PROGRAM P2_06_Device_Ctrl
VAR
	fbMixer_Motor					:FB_MotorFreqCtrl;
	fbMixerMotor_Speed				:FB_AnalogOutput_v01;
	fbSieve_Motor					:FB_MotorFreqCtrl;
	fbSieveMotor_Speed				:FB_AnalogOutput_v01;
	fbChopper_Motor					:FB_MotorCoilsCtrl;
	fbPump_Motor					:FB_CoilCtrl;
	
	fbSP_Temperature_PID			:FB_PID;
	
	fbSP_Mixer_Motor				:FB_MotorFreqCtrl;
	fbSP_MixerMotor_Speed			:FB_AnalogOutput_v01;
	fbSP_Pressure					:FB_AnalogOutput_v02;
	
	fbOutlet_Valve					:FB_ValveCtrl52;
	fbLid_Valve						:FB_ValveCtrl52;
	fbSieveSeal_Valve				:FB_ValveCtrl52;
	fbPurge_Valve					:FB_ValveCtrl52;
	fbTool_Valve					:FB_ValveCtrl52;
	
	fbCleaningAir_Valve				:FB_ValveCtrl32;
	fbPurifiedWater_Valve			:FB_ValveCtrl32;
	fbWarmWater_Valve				:FB_ValveCtrl32;
	fbColdWater_Valve				:FB_ValveCtrl32;
	fbMixerWIP_Valve				:FB_ValveCtrl32;
	fbChopperWIP_Valve				:FB_ValveCtrl32;
	fbSPWIP_Valve					:FB_ValveCtrl32;
	fbSPWIPDrain_Valve				:FB_ValveCtrl32;
	fbMainDrain_Valve				:FB_ValveCtrl32;
	
	fbAspiration_Valve				:FB_ValveCtrl32;
	fbVacuum_Valve					:FB_ValveCtrl32;
	fbFilterClean_Valve				:FB_ValveCtrl32;
	fbAirSeal_Valve					:FB_ValveCtrl32;
	fbMixerAir_Valve				:FB_ValveCtrl32;
	fbChopperAir_Valve				:FB_ValveCtrl32;
	
	
	
	

END_VAR

VAR PERSISTENT
	stMixer_Motor_Int				:ST_Interface_MotorCtrl;
	stSieve_Motor_Int				:ST_Interface_MotorCtrl;
	stChopper_Motor_Int				:ST_Interface_MotorCoilsCtrl;
	stPump_Motor_Int				:ST_Interface_CoilCtrl;
	
	stSP_Mixer_Motor_Int			:ST_Interface_MotorCtrl;
	stSP_Temperature_Int			:ST_Interface_PidCtrl;
	
	stOutlet_Valve_Int				:ST_Interface_ValveCtrl;
	stLid_Valve_Int					:ST_Interface_ValveCtrl;
	stSeal_Valve_Int				:ST_Interface_ValveCtrl;
	stPurge_Valve_Int				:ST_Interface_ValveCtrl;
	stTool_Valve_Int				:ST_Interface_ValveCtrl;
	
	stCleaningAir_Valve_INT			:ST_Interface_ValveCtrl;
	stPurifiedWater_Valve_INT		:ST_Interface_ValveCtrl;
	stWarmWater_Valve_Int			:ST_Interface_ValveCtrl;
	stColdWater_Valve_Int			:ST_Interface_ValveCtrl;
	stMixerWIP_Valve_Int			:ST_Interface_ValveCtrl;
	stChopperWIP_Valve_Int			:ST_Interface_ValveCtrl;
	stSPWIP_Valve_Int				:ST_Interface_ValveCtrl;
	stSPWIPDrain_Valve_Int			:ST_Interface_ValveCtrl;
	stMainDrain_Valve_Int			:ST_Interface_ValveCtrl;
	
	stAspiration_Valve_Int			:ST_Interface_ValveCtrl;
	stVacuum_Valve_Int				:ST_Interface_ValveCtrl;
	stFilterClean_Valve_Int			:ST_Interface_ValveCtrl;
	stAirSeal_Valve_Int				:ST_Interface_ValveCtrl;
	stMixerAir_Valve_Int			:ST_Interface_ValveCtrl;
	stChopperAir_Valve_Int			:ST_Interface_ValveCtrl;
END_VAR
VAR // added by the converter: edge detectors and wires of the graphical bodies
    _w1, _w2, _w3, _w4, _w5, _w6, _w7, _w8, _w9, _w10 : BOOL;
    _rt1, _rt2 : R_TRIG;
END_VAR

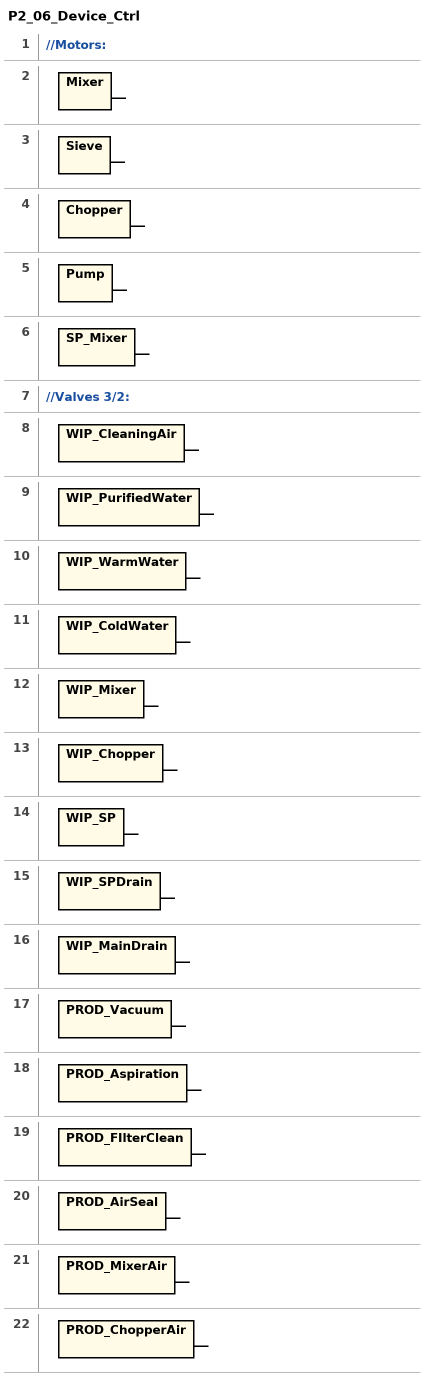
// NETWORK 1
// label: //Motors

// NETWORK 2
Mixer();

// NETWORK 3
Sieve();

// NETWORK 4
Chopper();

// NETWORK 5
Pump();

// NETWORK 6
SP_Mixer();

// NETWORK 7
// label: //Valves 3/2

// NETWORK 8
WIP_CleaningAir();

// NETWORK 9
WIP_PurifiedWater();

// NETWORK 10
WIP_WarmWater();

// NETWORK 11
WIP_ColdWater();

// NETWORK 12
WIP_Mixer();

// NETWORK 13
WIP_Chopper();

// NETWORK 14
WIP_SP();

// NETWORK 15
WIP_SPDrain();

// NETWORK 16
WIP_MainDrain();

// NETWORK 17
PROD_Vacuum();

// NETWORK 18
PROD_Aspiration();

// NETWORK 19
PROD_FIlterClean();

// NETWORK 20
PROD_AirSeal();

// NETWORK 21
PROD_MixerAir();

// NETWORK 22
PROD_ChopperAir();

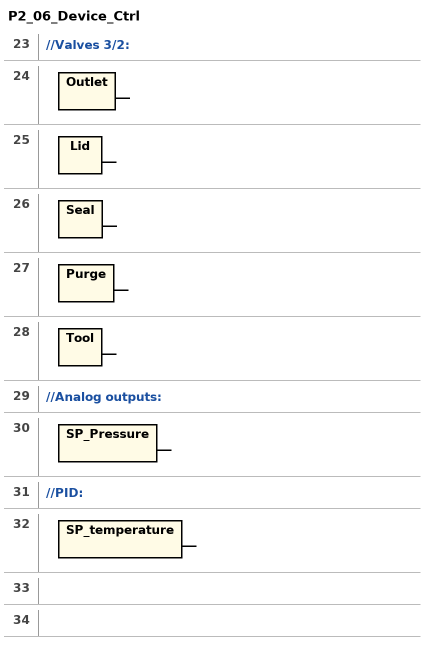
// NETWORK 23
// label: //Valves 3/2

// NETWORK 24
Outlet();

// NETWORK 25
Lid();

// NETWORK 26
Seal();

// NETWORK 27
Purge();

// NETWORK 28
Tool();

// NETWORK 29
// label: //Analog outputs

// NETWORK 30
SP_Pressure();

// NETWORK 31
// label: //PID

// NETWORK 32
SP_temperature();

// NETWORK 33

// NETWORK 34

ACTION Chopper:
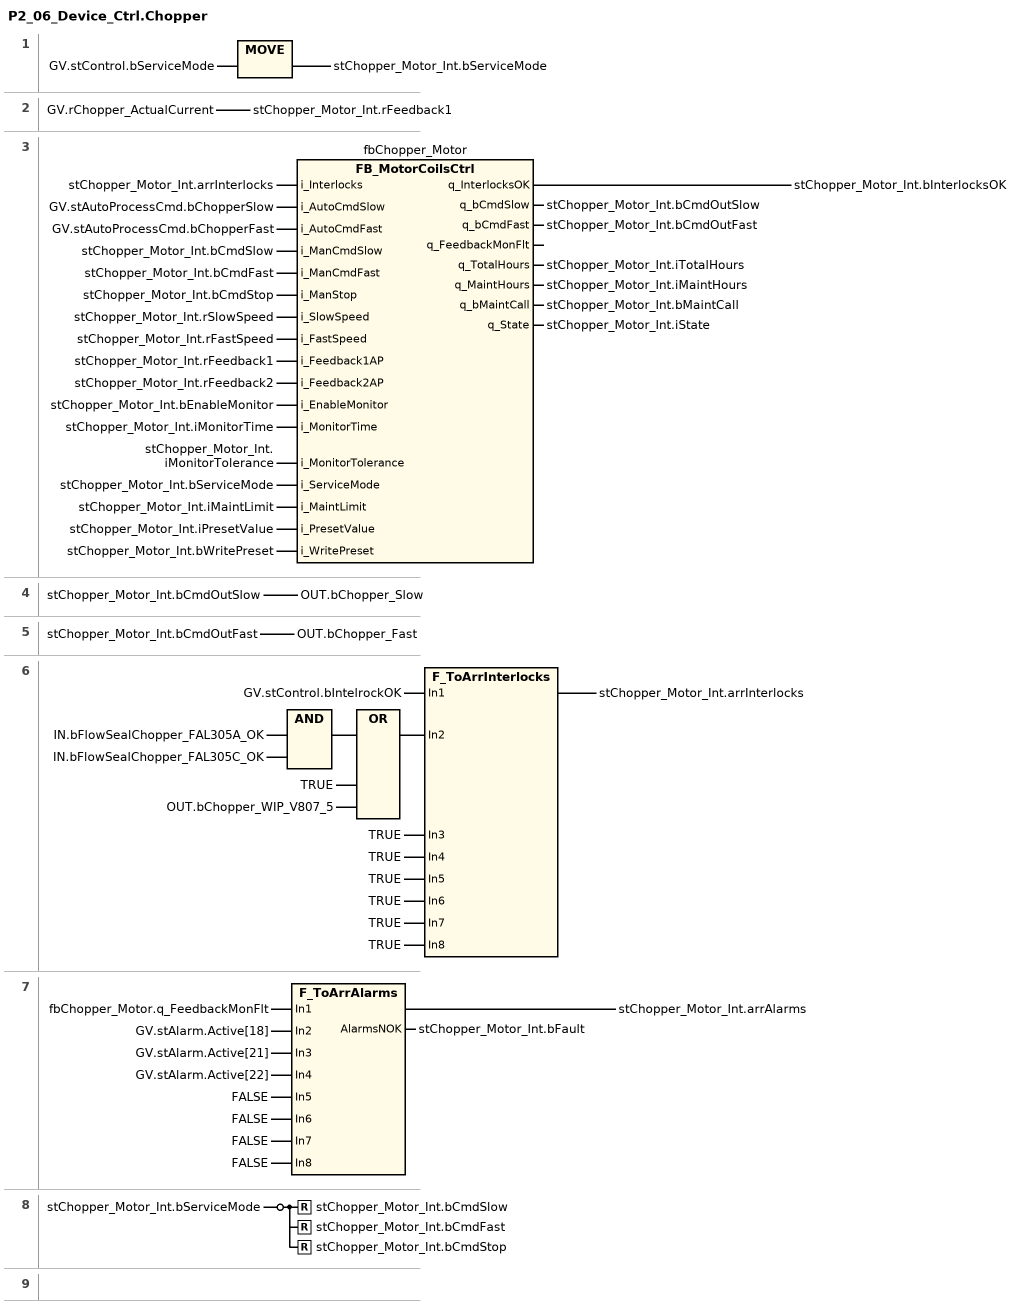
// NETWORK 1
stChopper_Motor_Int.bServiceMode := GV.stControl.bServiceMode;

// NETWORK 2
stChopper_Motor_Int.rFeedback1 := GV.rChopper_ActualCurrent;

// NETWORK 3
fbChopper_Motor(
    i_Interlocks := stChopper_Motor_Int.arrInterlocks,
    i_AutoCmdSlow := GV.stAutoProcessCmd.bChopperSlow,
    i_AutoCmdFast := GV.stAutoProcessCmd.bChopperFast,
    i_ManCmdSlow := stChopper_Motor_Int.bCmdSlow,
    i_ManCmdFast := stChopper_Motor_Int.bCmdFast,
    i_ManStop := stChopper_Motor_Int.bCmdStop,
    i_SlowSpeed := stChopper_Motor_Int.rSlowSpeed,
    i_FastSpeed := stChopper_Motor_Int.rFastSpeed,
    i_Feedback1AP := stChopper_Motor_Int.rFeedback1,
    i_Feedback2AP := stChopper_Motor_Int.rFeedback2,
    i_EnableMonitor := stChopper_Motor_Int.bEnableMonitor,
    i_MonitorTime := stChopper_Motor_Int.iMonitorTime,
    i_MonitorTolerance := stChopper_Motor_Int.iMonitorTolerance,
    i_ServiceMode := stChopper_Motor_Int.bServiceMode,
    i_MaintLimit := stChopper_Motor_Int.iMaintLimit,
    i_PresetValue := stChopper_Motor_Int.iPresetValue,
    i_WritePreset := stChopper_Motor_Int.bWritePreset,
    q_bCmdSlow => stChopper_Motor_Int.bCmdOutSlow,
    q_bCmdFast => stChopper_Motor_Int.bCmdOutFast,
    q_TotalHours => stChopper_Motor_Int.iTotalHours,
    q_MaintHours => stChopper_Motor_Int.iMaintHours,
    q_bMaintCall => stChopper_Motor_Int.bMaintCall,
    q_State => stChopper_Motor_Int.iState); // FB_MotorCoilsCtrl
stChopper_Motor_Int.bInterlocksOK := fbChopper_Motor.q_InterlocksOK;

// NETWORK 4
OUT.bChopper_Slow := stChopper_Motor_Int.bCmdOutSlow;

// NETWORK 5
OUT.bChopper_Fast := stChopper_Motor_Int.bCmdOutFast;

// NETWORK 6
stChopper_Motor_Int.arrInterlocks := F_ToArrInterlocks(In1 := GV.stControl.bIntelrockOK, In2 := IN.bFlowSealChopper_FAL305A_OK AND IN.bFlowSealChopper_FAL305C_OK OR TRUE OR OUT.bChopper_WIP_V807_5, In3 := TRUE, In4 := TRUE, In5 := TRUE, In6 := TRUE, In7 := TRUE, In8 := TRUE);

// NETWORK 7
stChopper_Motor_Int.arrAlarms := F_ToArrAlarms(In1 := fbChopper_Motor.q_FeedbackMonFlt, In2 := GV.stAlarm.Active[18], In3 := GV.stAlarm.Active[21], In4 := GV.stAlarm.Active[22], In5 := FALSE, In6 := FALSE, In7 := FALSE, In8 := FALSE, AlarmsNOK => stChopper_Motor_Int.bFault);

// NETWORK 8
_w1 := NOT stChopper_Motor_Int.bServiceMode;
stChopper_Motor_Int.bCmdSlow R= _w1;
stChopper_Motor_Int.bCmdFast R= _w1;
stChopper_Motor_Int.bCmdStop R= _w1;

// NETWORK 9
END_ACTION

ACTION Lid:
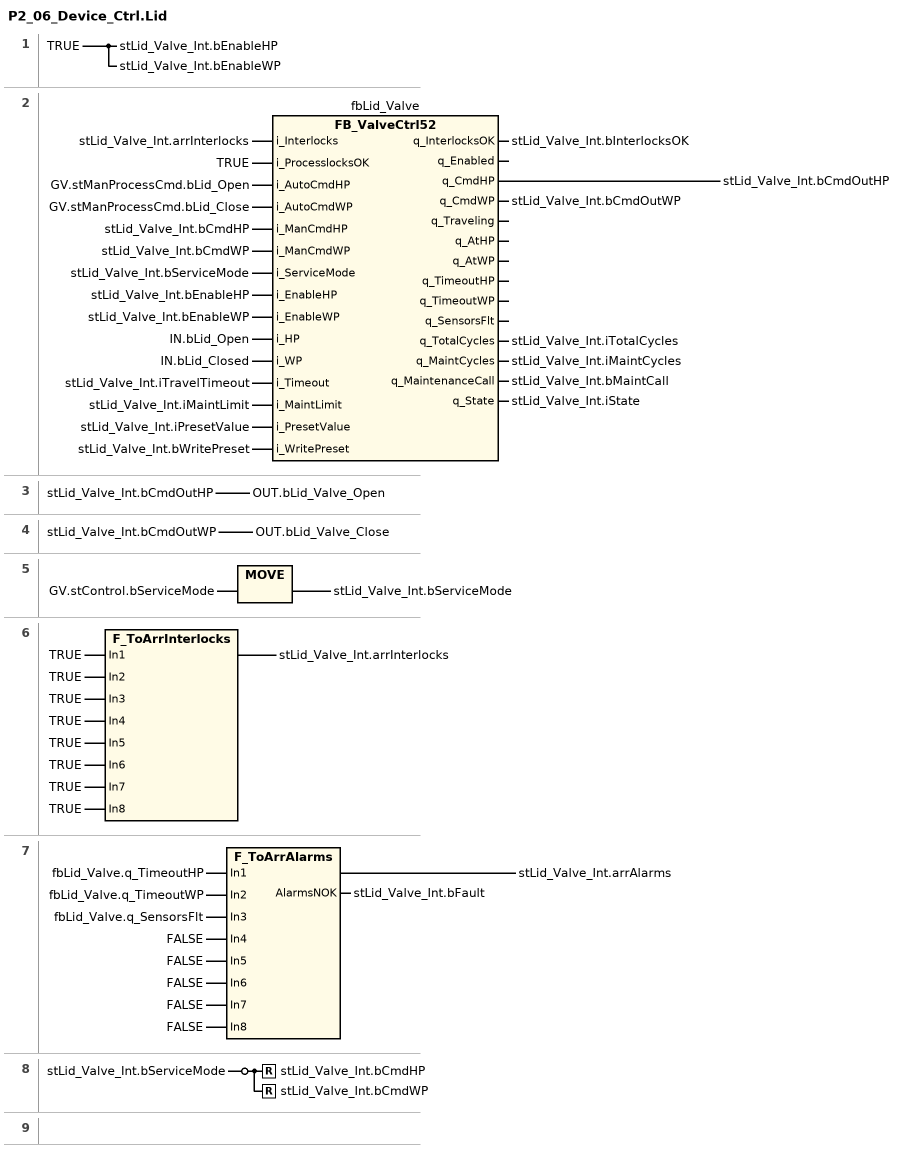
// NETWORK 1
stLid_Valve_Int.bEnableHP := TRUE;
stLid_Valve_Int.bEnableWP := TRUE;

// NETWORK 2
fbLid_Valve(
    i_Interlocks := stLid_Valve_Int.arrInterlocks,
    i_ProcesslocksOK := TRUE,
    i_AutoCmdHP := GV.stManProcessCmd.bLid_Open,
    i_AutoCmdWP := GV.stManProcessCmd.bLid_Close,
    i_ManCmdHP := stLid_Valve_Int.bCmdHP,
    i_ManCmdWP := stLid_Valve_Int.bCmdWP,
    i_ServiceMode := stLid_Valve_Int.bServiceMode,
    i_EnableHP := stLid_Valve_Int.bEnableHP,
    i_EnableWP := stLid_Valve_Int.bEnableWP,
    i_HP := IN.bLid_Open,
    i_WP := IN.bLid_Closed,
    i_Timeout := stLid_Valve_Int.iTravelTimeout,
    i_MaintLimit := stLid_Valve_Int.iMaintLimit,
    i_PresetValue := stLid_Valve_Int.iPresetValue,
    i_WritePreset := stLid_Valve_Int.bWritePreset,
    q_InterlocksOK => stLid_Valve_Int.bInterlocksOK,
    q_CmdWP => stLid_Valve_Int.bCmdOutWP,
    q_TotalCycles => stLid_Valve_Int.iTotalCycles,
    q_MaintCycles => stLid_Valve_Int.iMaintCycles,
    q_MaintenanceCall => stLid_Valve_Int.bMaintCall,
    q_State => stLid_Valve_Int.iState); // FB_ValveCtrl52
stLid_Valve_Int.bCmdOutHP := fbLid_Valve.q_CmdHP;

// NETWORK 3
OUT.bLid_Valve_Open := stLid_Valve_Int.bCmdOutHP;

// NETWORK 4
OUT.bLid_Valve_Close := stLid_Valve_Int.bCmdOutWP;

// NETWORK 5
stLid_Valve_Int.bServiceMode := GV.stControl.bServiceMode;

// NETWORK 6
stLid_Valve_Int.arrInterlocks := F_ToArrInterlocks(In1 := TRUE, In2 := TRUE, In3 := TRUE, In4 := TRUE, In5 := TRUE, In6 := TRUE, In7 := TRUE, In8 := TRUE);

// NETWORK 7
stLid_Valve_Int.arrAlarms := F_ToArrAlarms(In1 := fbLid_Valve.q_TimeoutHP, In2 := fbLid_Valve.q_TimeoutWP, In3 := fbLid_Valve.q_SensorsFlt, In4 := FALSE, In5 := FALSE, In6 := FALSE, In7 := FALSE, In8 := FALSE, AlarmsNOK => stLid_Valve_Int.bFault);

// NETWORK 8
_w2 := NOT stLid_Valve_Int.bServiceMode;
stLid_Valve_Int.bCmdHP R= _w2;
stLid_Valve_Int.bCmdWP R= _w2;

// NETWORK 9
END_ACTION

ACTION Mixer:
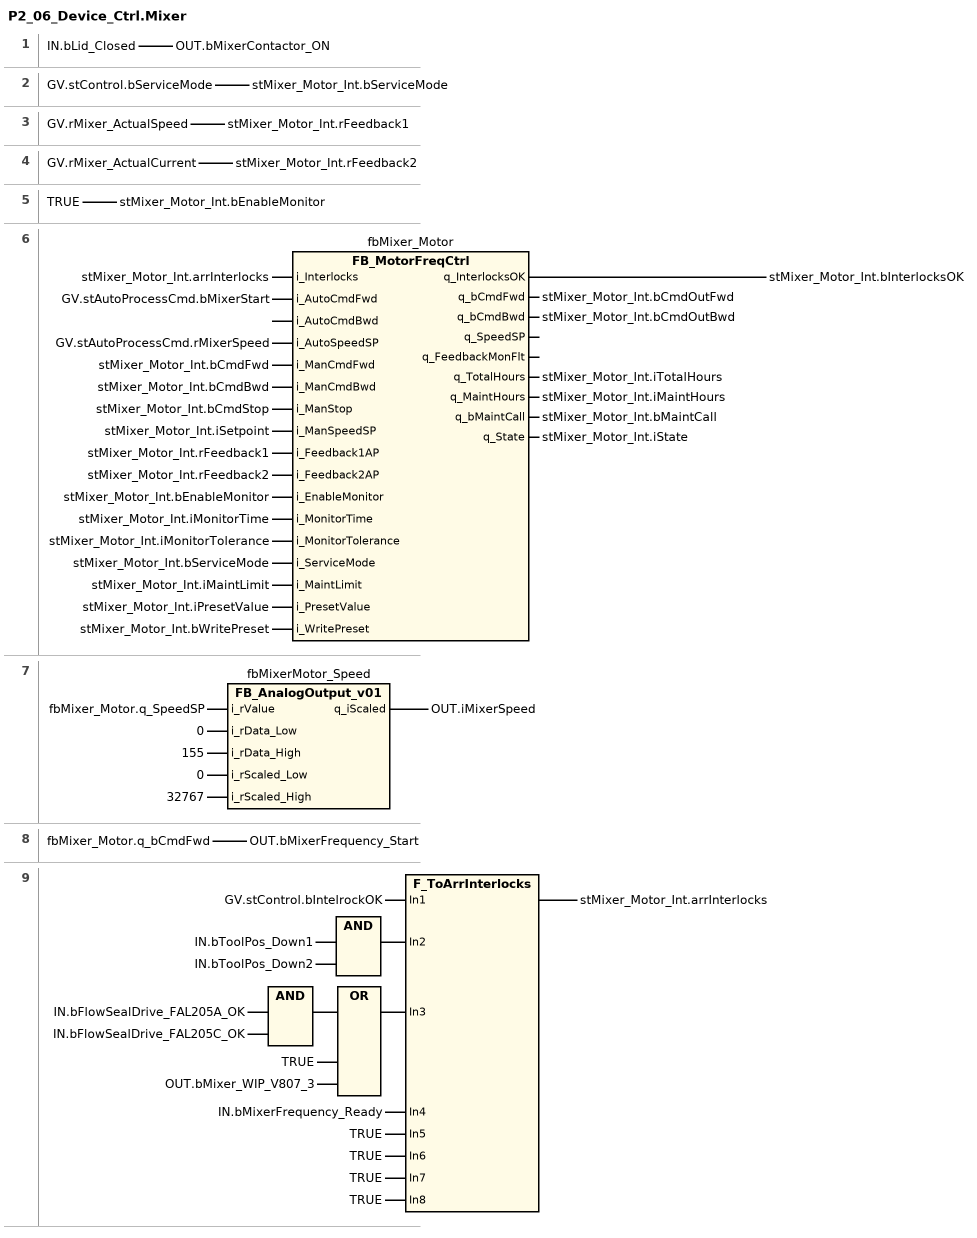
// NETWORK 1
OUT.bMixerContactor_ON := IN.bLid_Closed;

// NETWORK 2
stMixer_Motor_Int.bServiceMode := GV.stControl.bServiceMode;

// NETWORK 3
stMixer_Motor_Int.rFeedback1 := GV.rMixer_ActualSpeed;

// NETWORK 4
stMixer_Motor_Int.rFeedback2 := GV.rMixer_ActualCurrent;

// NETWORK 5
stMixer_Motor_Int.bEnableMonitor := TRUE;

// NETWORK 6
fbMixer_Motor(
    i_Interlocks := stMixer_Motor_Int.arrInterlocks,
    i_AutoCmdFwd := GV.stAutoProcessCmd.bMixerStart,
    i_AutoSpeedSP := GV.stAutoProcessCmd.rMixerSpeed,
    i_ManCmdFwd := stMixer_Motor_Int.bCmdFwd,
    i_ManCmdBwd := stMixer_Motor_Int.bCmdBwd,
    i_ManStop := stMixer_Motor_Int.bCmdStop,
    i_ManSpeedSP := stMixer_Motor_Int.iSetpoint,
    i_Feedback1AP := stMixer_Motor_Int.rFeedback1,
    i_Feedback2AP := stMixer_Motor_Int.rFeedback2,
    i_EnableMonitor := stMixer_Motor_Int.bEnableMonitor,
    i_MonitorTime := stMixer_Motor_Int.iMonitorTime,
    i_MonitorTolerance := stMixer_Motor_Int.iMonitorTolerance,
    i_ServiceMode := stMixer_Motor_Int.bServiceMode,
    i_MaintLimit := stMixer_Motor_Int.iMaintLimit,
    i_PresetValue := stMixer_Motor_Int.iPresetValue,
    i_WritePreset := stMixer_Motor_Int.bWritePreset,
    q_bCmdFwd => stMixer_Motor_Int.bCmdOutFwd,
    q_bCmdBwd => stMixer_Motor_Int.bCmdOutBwd,
    q_TotalHours => stMixer_Motor_Int.iTotalHours,
    q_MaintHours => stMixer_Motor_Int.iMaintHours,
    q_bMaintCall => stMixer_Motor_Int.bMaintCall,
    q_State => stMixer_Motor_Int.iState); // FB_MotorFreqCtrl
stMixer_Motor_Int.bInterlocksOK := fbMixer_Motor.q_InterlocksOK;

// NETWORK 7
fbMixerMotor_Speed(
    i_rValue := fbMixer_Motor.q_SpeedSP,
    i_rData_Low := 0,
    i_rData_High := 155,
    i_rScaled_Low := 0,
    i_rScaled_High := 32767); // FB_AnalogOutput_v01
OUT.iMixerSpeed := fbMixerMotor_Speed.q_iScaled;

// NETWORK 8
OUT.bMixerFrequency_Start := fbMixer_Motor.q_bCmdFwd;

// NETWORK 9
stMixer_Motor_Int.arrInterlocks := F_ToArrInterlocks(In1 := GV.stControl.bIntelrockOK, In2 := IN.bToolPos_Down1 AND IN.bToolPos_Down2, In3 := IN.bFlowSealDrive_FAL205A_OK AND IN.bFlowSealDrive_FAL205C_OK OR TRUE OR OUT.bMixer_WIP_V807_3, In4 := IN.bMixerFrequency_Ready, In5 := TRUE, In6 := TRUE, In7 := TRUE, In8 := TRUE);

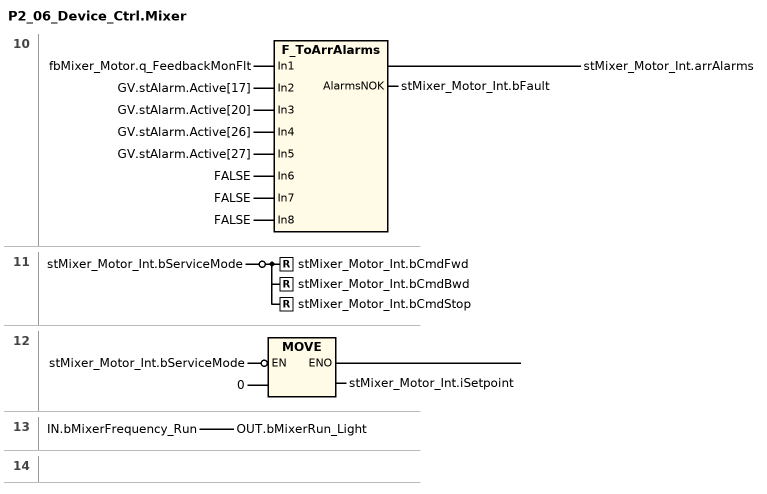
// NETWORK 10
stMixer_Motor_Int.arrAlarms := F_ToArrAlarms(In1 := fbMixer_Motor.q_FeedbackMonFlt, In2 := GV.stAlarm.Active[17], In3 := GV.stAlarm.Active[20], In4 := GV.stAlarm.Active[26], In5 := GV.stAlarm.Active[27], In6 := FALSE, In7 := FALSE, In8 := FALSE, AlarmsNOK => stMixer_Motor_Int.bFault);

// NETWORK 11
_w3 := NOT stMixer_Motor_Int.bServiceMode;
stMixer_Motor_Int.bCmdFwd R= _w3;
stMixer_Motor_Int.bCmdBwd R= _w3;
stMixer_Motor_Int.bCmdStop R= _w3;

// NETWORK 12
IF NOT stMixer_Motor_Int.bServiceMode THEN stMixer_Motor_Int.iSetpoint := 0; END_IF

// NETWORK 13
OUT.bMixerRun_Light := IN.bMixerFrequency_Run;

// NETWORK 14
END_ACTION

ACTION Outlet:
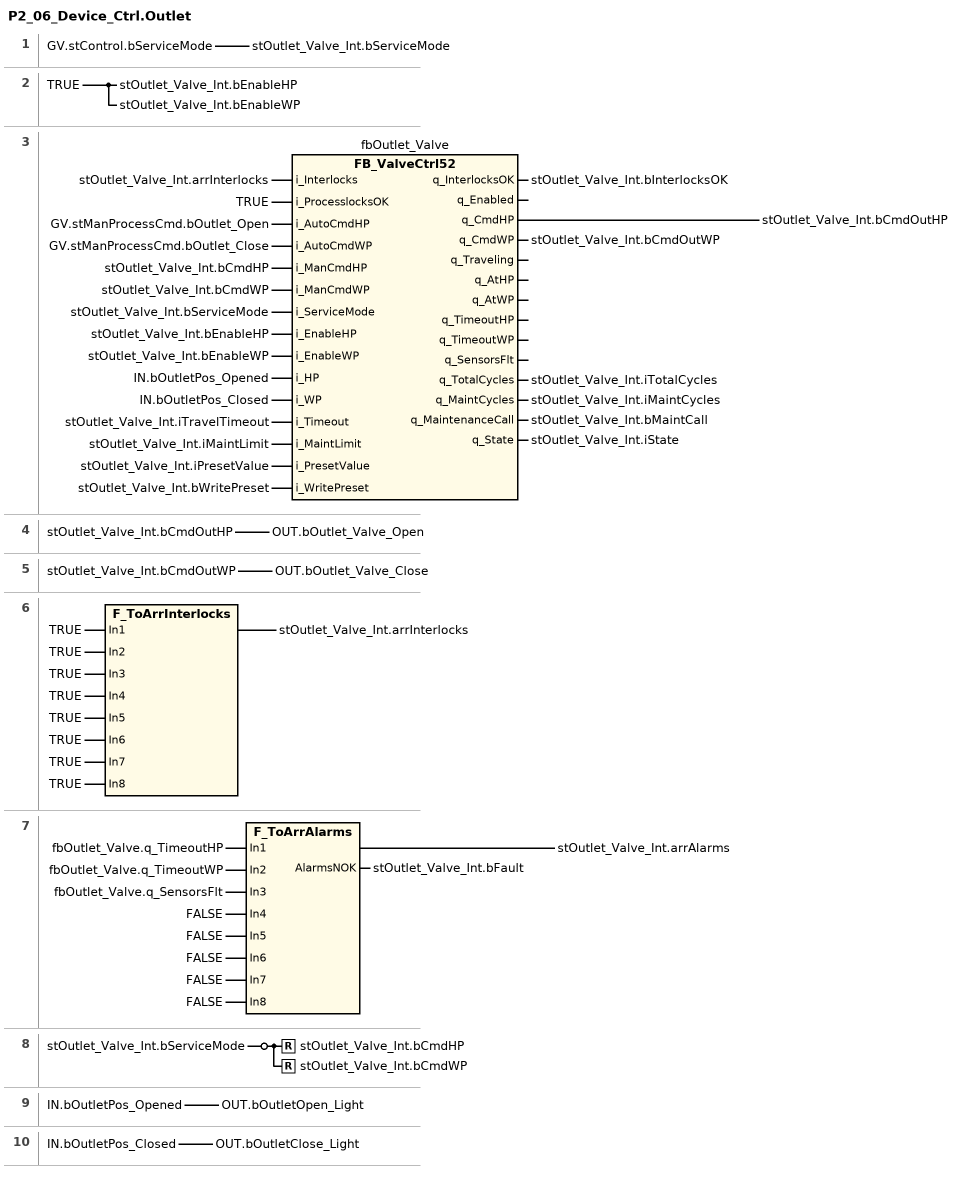
// NETWORK 1
stOutlet_Valve_Int.bServiceMode := GV.stControl.bServiceMode;

// NETWORK 2
stOutlet_Valve_Int.bEnableHP := TRUE;
stOutlet_Valve_Int.bEnableWP := TRUE;

// NETWORK 3
fbOutlet_Valve(
    i_Interlocks := stOutlet_Valve_Int.arrInterlocks,
    i_ProcesslocksOK := TRUE,
    i_AutoCmdHP := GV.stManProcessCmd.bOutlet_Open,
    i_AutoCmdWP := GV.stManProcessCmd.bOutlet_Close,
    i_ManCmdHP := stOutlet_Valve_Int.bCmdHP,
    i_ManCmdWP := stOutlet_Valve_Int.bCmdWP,
    i_ServiceMode := stOutlet_Valve_Int.bServiceMode,
    i_EnableHP := stOutlet_Valve_Int.bEnableHP,
    i_EnableWP := stOutlet_Valve_Int.bEnableWP,
    i_HP := IN.bOutletPos_Opened,
    i_WP := IN.bOutletPos_Closed,
    i_Timeout := stOutlet_Valve_Int.iTravelTimeout,
    i_MaintLimit := stOutlet_Valve_Int.iMaintLimit,
    i_PresetValue := stOutlet_Valve_Int.iPresetValue,
    i_WritePreset := stOutlet_Valve_Int.bWritePreset,
    q_InterlocksOK => stOutlet_Valve_Int.bInterlocksOK,
    q_CmdWP => stOutlet_Valve_Int.bCmdOutWP,
    q_TotalCycles => stOutlet_Valve_Int.iTotalCycles,
    q_MaintCycles => stOutlet_Valve_Int.iMaintCycles,
    q_MaintenanceCall => stOutlet_Valve_Int.bMaintCall,
    q_State => stOutlet_Valve_Int.iState); // FB_ValveCtrl52
stOutlet_Valve_Int.bCmdOutHP := fbOutlet_Valve.q_CmdHP;

// NETWORK 4
OUT.bOutlet_Valve_Open := stOutlet_Valve_Int.bCmdOutHP;

// NETWORK 5
OUT.bOutlet_Valve_Close := stOutlet_Valve_Int.bCmdOutWP;

// NETWORK 6
stOutlet_Valve_Int.arrInterlocks := F_ToArrInterlocks(In1 := TRUE, In2 := TRUE, In3 := TRUE, In4 := TRUE, In5 := TRUE, In6 := TRUE, In7 := TRUE, In8 := TRUE);

// NETWORK 7
stOutlet_Valve_Int.arrAlarms := F_ToArrAlarms(In1 := fbOutlet_Valve.q_TimeoutHP, In2 := fbOutlet_Valve.q_TimeoutWP, In3 := fbOutlet_Valve.q_SensorsFlt, In4 := FALSE, In5 := FALSE, In6 := FALSE, In7 := FALSE, In8 := FALSE, AlarmsNOK => stOutlet_Valve_Int.bFault);

// NETWORK 8
_w4 := NOT stOutlet_Valve_Int.bServiceMode;
stOutlet_Valve_Int.bCmdHP R= _w4;
stOutlet_Valve_Int.bCmdWP R= _w4;

// NETWORK 9
OUT.bOutletOpen_Light := IN.bOutletPos_Opened;

// NETWORK 10
OUT.bOutletClose_Light := IN.bOutletPos_Closed;
END_ACTION

ACTION PROD_AirSeal:
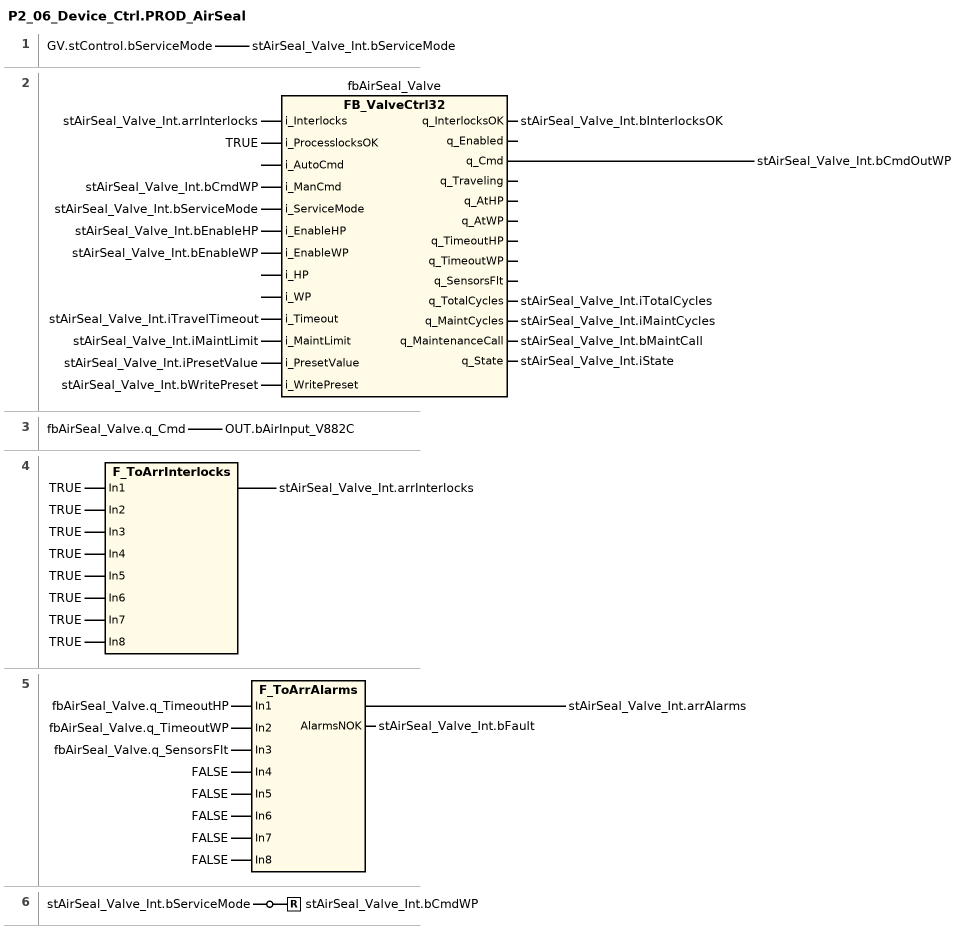
// NETWORK 1
stAirSeal_Valve_Int.bServiceMode := GV.stControl.bServiceMode;

// NETWORK 2
fbAirSeal_Valve(
    i_Interlocks := stAirSeal_Valve_Int.arrInterlocks,
    i_ProcesslocksOK := TRUE,
    i_ManCmd := stAirSeal_Valve_Int.bCmdWP,
    i_ServiceMode := stAirSeal_Valve_Int.bServiceMode,
    i_EnableHP := stAirSeal_Valve_Int.bEnableHP,
    i_EnableWP := stAirSeal_Valve_Int.bEnableWP,
    i_Timeout := stAirSeal_Valve_Int.iTravelTimeout,
    i_MaintLimit := stAirSeal_Valve_Int.iMaintLimit,
    i_PresetValue := stAirSeal_Valve_Int.iPresetValue,
    i_WritePreset := stAirSeal_Valve_Int.bWritePreset,
    q_InterlocksOK => stAirSeal_Valve_Int.bInterlocksOK,
    q_TotalCycles => stAirSeal_Valve_Int.iTotalCycles,
    q_MaintCycles => stAirSeal_Valve_Int.iMaintCycles,
    q_MaintenanceCall => stAirSeal_Valve_Int.bMaintCall,
    q_State => stAirSeal_Valve_Int.iState); // FB_ValveCtrl32
stAirSeal_Valve_Int.bCmdOutWP := fbAirSeal_Valve.q_Cmd;

// NETWORK 3
OUT.bAirInput_V882C := fbAirSeal_Valve.q_Cmd;

// NETWORK 4
stAirSeal_Valve_Int.arrInterlocks := F_ToArrInterlocks(In1 := TRUE, In2 := TRUE, In3 := TRUE, In4 := TRUE, In5 := TRUE, In6 := TRUE, In7 := TRUE, In8 := TRUE);

// NETWORK 5
stAirSeal_Valve_Int.arrAlarms := F_ToArrAlarms(In1 := fbAirSeal_Valve.q_TimeoutHP, In2 := fbAirSeal_Valve.q_TimeoutWP, In3 := fbAirSeal_Valve.q_SensorsFlt, In4 := FALSE, In5 := FALSE, In6 := FALSE, In7 := FALSE, In8 := FALSE, AlarmsNOK => stAirSeal_Valve_Int.bFault);

// NETWORK 6
stAirSeal_Valve_Int.bCmdWP R= NOT stAirSeal_Valve_Int.bServiceMode;
END_ACTION

ACTION PROD_Aspiration:
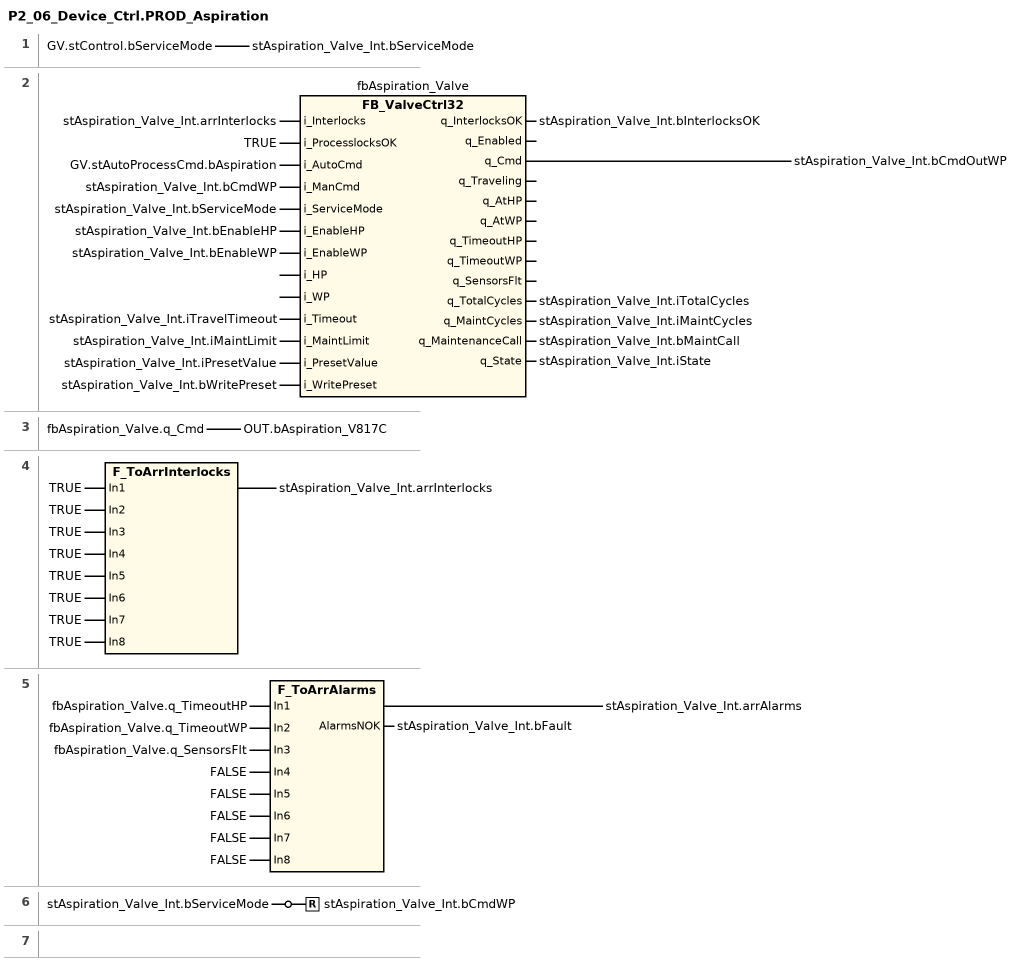
// NETWORK 1
stAspiration_Valve_Int.bServiceMode := GV.stControl.bServiceMode;

// NETWORK 2
fbAspiration_Valve(
    i_Interlocks := stAspiration_Valve_Int.arrInterlocks,
    i_ProcesslocksOK := TRUE,
    i_AutoCmd := GV.stAutoProcessCmd.bAspiration,
    i_ManCmd := stAspiration_Valve_Int.bCmdWP,
    i_ServiceMode := stAspiration_Valve_Int.bServiceMode,
    i_EnableHP := stAspiration_Valve_Int.bEnableHP,
    i_EnableWP := stAspiration_Valve_Int.bEnableWP,
    i_Timeout := stAspiration_Valve_Int.iTravelTimeout,
    i_MaintLimit := stAspiration_Valve_Int.iMaintLimit,
    i_PresetValue := stAspiration_Valve_Int.iPresetValue,
    i_WritePreset := stAspiration_Valve_Int.bWritePreset,
    q_InterlocksOK => stAspiration_Valve_Int.bInterlocksOK,
    q_TotalCycles => stAspiration_Valve_Int.iTotalCycles,
    q_MaintCycles => stAspiration_Valve_Int.iMaintCycles,
    q_MaintenanceCall => stAspiration_Valve_Int.bMaintCall,
    q_State => stAspiration_Valve_Int.iState); // FB_ValveCtrl32
stAspiration_Valve_Int.bCmdOutWP := fbAspiration_Valve.q_Cmd;

// NETWORK 3
OUT.bAspiration_V817C := fbAspiration_Valve.q_Cmd;

// NETWORK 4
stAspiration_Valve_Int.arrInterlocks := F_ToArrInterlocks(In1 := TRUE, In2 := TRUE, In3 := TRUE, In4 := TRUE, In5 := TRUE, In6 := TRUE, In7 := TRUE, In8 := TRUE);

// NETWORK 5
stAspiration_Valve_Int.arrAlarms := F_ToArrAlarms(In1 := fbAspiration_Valve.q_TimeoutHP, In2 := fbAspiration_Valve.q_TimeoutWP, In3 := fbAspiration_Valve.q_SensorsFlt, In4 := FALSE, In5 := FALSE, In6 := FALSE, In7 := FALSE, In8 := FALSE, AlarmsNOK => stAspiration_Valve_Int.bFault);

// NETWORK 6
stAspiration_Valve_Int.bCmdWP R= NOT stAspiration_Valve_Int.bServiceMode;

// NETWORK 7
END_ACTION

ACTION PROD_ChopperAir:
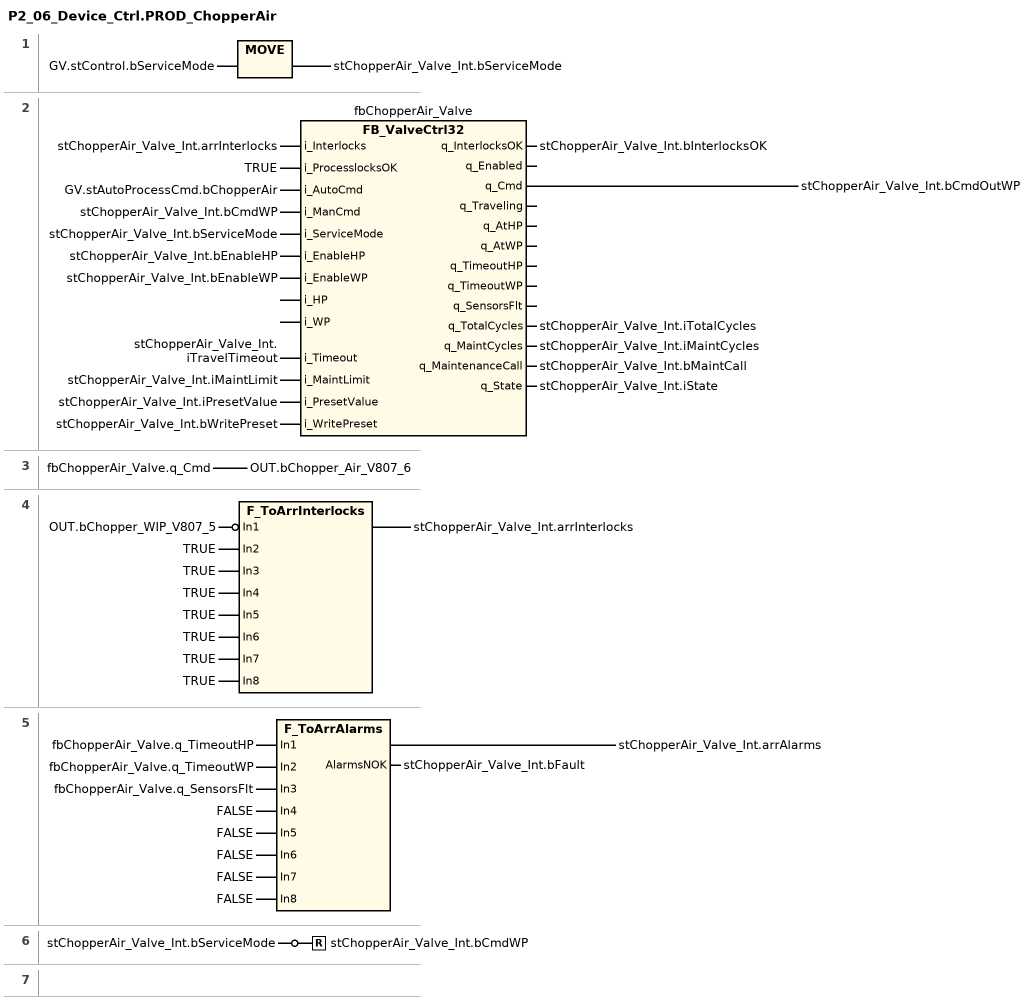
// NETWORK 1
stChopperAir_Valve_Int.bServiceMode := GV.stControl.bServiceMode;

// NETWORK 2
fbChopperAir_Valve(
    i_Interlocks := stChopperAir_Valve_Int.arrInterlocks,
    i_ProcesslocksOK := TRUE,
    i_AutoCmd := GV.stAutoProcessCmd.bChopperAir,
    i_ManCmd := stChopperAir_Valve_Int.bCmdWP,
    i_ServiceMode := stChopperAir_Valve_Int.bServiceMode,
    i_EnableHP := stChopperAir_Valve_Int.bEnableHP,
    i_EnableWP := stChopperAir_Valve_Int.bEnableWP,
    i_Timeout := stChopperAir_Valve_Int.iTravelTimeout,
    i_MaintLimit := stChopperAir_Valve_Int.iMaintLimit,
    i_PresetValue := stChopperAir_Valve_Int.iPresetValue,
    i_WritePreset := stChopperAir_Valve_Int.bWritePreset,
    q_InterlocksOK => stChopperAir_Valve_Int.bInterlocksOK,
    q_TotalCycles => stChopperAir_Valve_Int.iTotalCycles,
    q_MaintCycles => stChopperAir_Valve_Int.iMaintCycles,
    q_MaintenanceCall => stChopperAir_Valve_Int.bMaintCall,
    q_State => stChopperAir_Valve_Int.iState); // FB_ValveCtrl32
stChopperAir_Valve_Int.bCmdOutWP := fbChopperAir_Valve.q_Cmd;

// NETWORK 3
OUT.bChopper_Air_V807_6 := fbChopperAir_Valve.q_Cmd;

// NETWORK 4
stChopperAir_Valve_Int.arrInterlocks := F_ToArrInterlocks(In1 := NOT OUT.bChopper_WIP_V807_5, In2 := TRUE, In3 := TRUE, In4 := TRUE, In5 := TRUE, In6 := TRUE, In7 := TRUE, In8 := TRUE);

// NETWORK 5
stChopperAir_Valve_Int.arrAlarms := F_ToArrAlarms(In1 := fbChopperAir_Valve.q_TimeoutHP, In2 := fbChopperAir_Valve.q_TimeoutWP, In3 := fbChopperAir_Valve.q_SensorsFlt, In4 := FALSE, In5 := FALSE, In6 := FALSE, In7 := FALSE, In8 := FALSE, AlarmsNOK => stChopperAir_Valve_Int.bFault);

// NETWORK 6
stChopperAir_Valve_Int.bCmdWP R= NOT stChopperAir_Valve_Int.bServiceMode;

// NETWORK 7
END_ACTION

ACTION PROD_FilterClean:
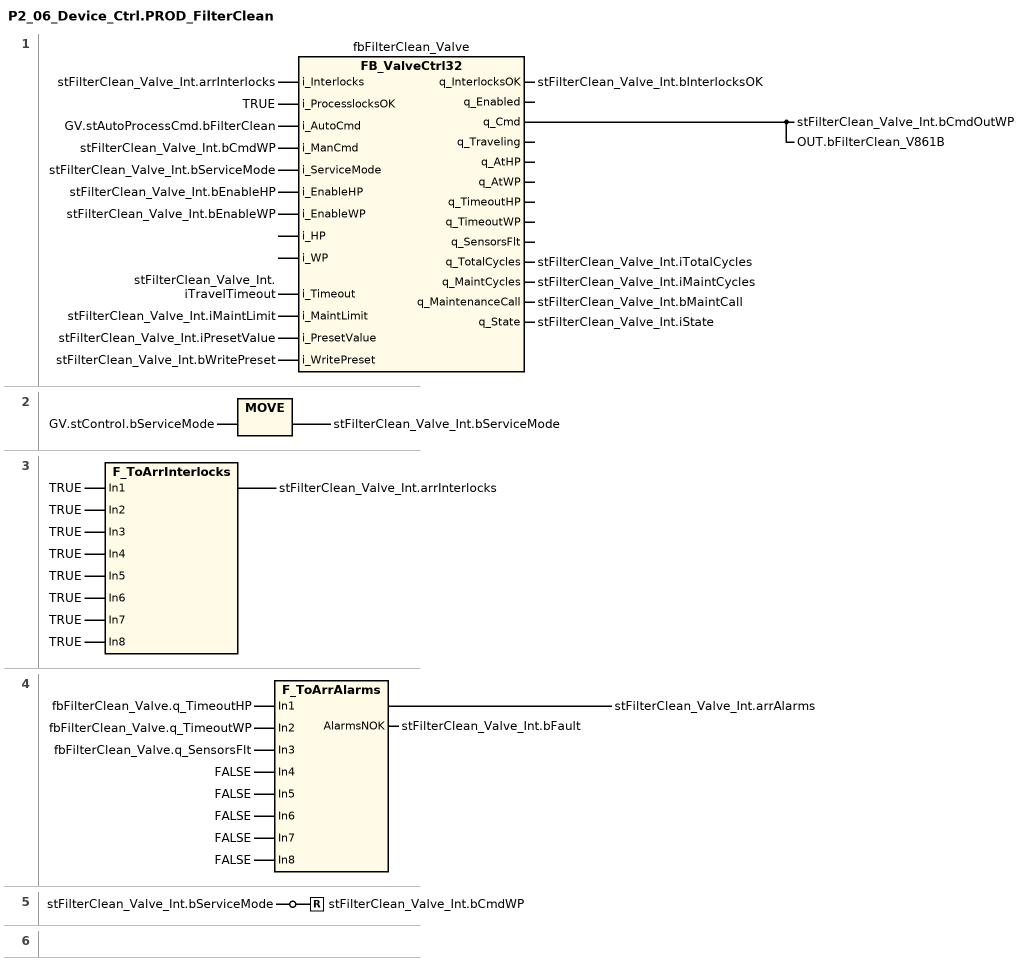
// NETWORK 1
fbFilterClean_Valve(
    i_Interlocks := stFilterClean_Valve_Int.arrInterlocks,
    i_ProcesslocksOK := TRUE,
    i_AutoCmd := GV.stAutoProcessCmd.bFilterClean,
    i_ManCmd := stFilterClean_Valve_Int.bCmdWP,
    i_ServiceMode := stFilterClean_Valve_Int.bServiceMode,
    i_EnableHP := stFilterClean_Valve_Int.bEnableHP,
    i_EnableWP := stFilterClean_Valve_Int.bEnableWP,
    i_Timeout := stFilterClean_Valve_Int.iTravelTimeout,
    i_MaintLimit := stFilterClean_Valve_Int.iMaintLimit,
    i_PresetValue := stFilterClean_Valve_Int.iPresetValue,
    i_WritePreset := stFilterClean_Valve_Int.bWritePreset,
    q_InterlocksOK => stFilterClean_Valve_Int.bInterlocksOK,
    q_TotalCycles => stFilterClean_Valve_Int.iTotalCycles,
    q_MaintCycles => stFilterClean_Valve_Int.iMaintCycles,
    q_MaintenanceCall => stFilterClean_Valve_Int.bMaintCall,
    q_State => stFilterClean_Valve_Int.iState); // FB_ValveCtrl32
stFilterClean_Valve_Int.bCmdOutWP := fbFilterClean_Valve.q_Cmd;
OUT.bFilterClean_V861B := fbFilterClean_Valve.q_Cmd;

// NETWORK 2
stFilterClean_Valve_Int.bServiceMode := GV.stControl.bServiceMode;

// NETWORK 3
stFilterClean_Valve_Int.arrInterlocks := F_ToArrInterlocks(In1 := TRUE, In2 := TRUE, In3 := TRUE, In4 := TRUE, In5 := TRUE, In6 := TRUE, In7 := TRUE, In8 := TRUE);

// NETWORK 4
stFilterClean_Valve_Int.arrAlarms := F_ToArrAlarms(In1 := fbFilterClean_Valve.q_TimeoutHP, In2 := fbFilterClean_Valve.q_TimeoutWP, In3 := fbFilterClean_Valve.q_SensorsFlt, In4 := FALSE, In5 := FALSE, In6 := FALSE, In7 := FALSE, In8 := FALSE, AlarmsNOK => stFilterClean_Valve_Int.bFault);

// NETWORK 5
stFilterClean_Valve_Int.bCmdWP R= NOT stFilterClean_Valve_Int.bServiceMode;

// NETWORK 6
END_ACTION

ACTION PROD_MixerAir:
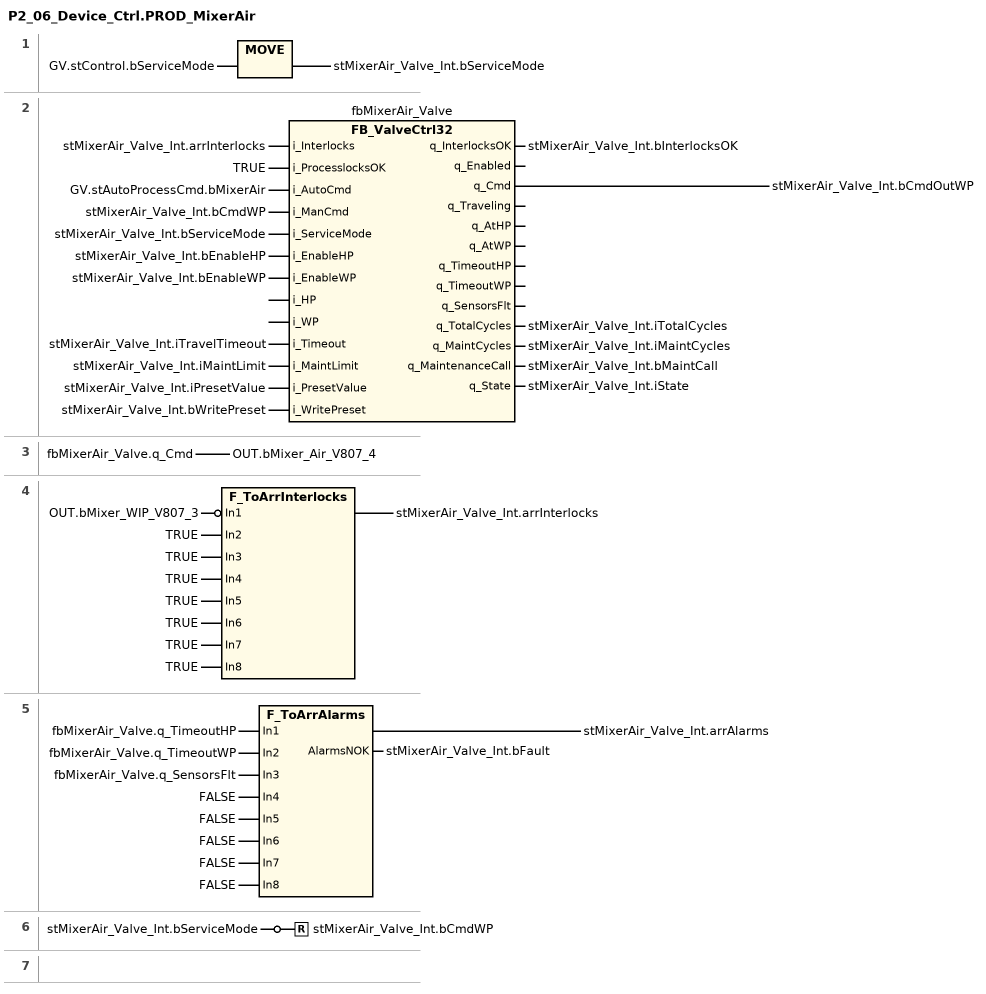
// NETWORK 1
stMixerAir_Valve_Int.bServiceMode := GV.stControl.bServiceMode;

// NETWORK 2
fbMixerAir_Valve(
    i_Interlocks := stMixerAir_Valve_Int.arrInterlocks,
    i_ProcesslocksOK := TRUE,
    i_AutoCmd := GV.stAutoProcessCmd.bMixerAir,
    i_ManCmd := stMixerAir_Valve_Int.bCmdWP,
    i_ServiceMode := stMixerAir_Valve_Int.bServiceMode,
    i_EnableHP := stMixerAir_Valve_Int.bEnableHP,
    i_EnableWP := stMixerAir_Valve_Int.bEnableWP,
    i_Timeout := stMixerAir_Valve_Int.iTravelTimeout,
    i_MaintLimit := stMixerAir_Valve_Int.iMaintLimit,
    i_PresetValue := stMixerAir_Valve_Int.iPresetValue,
    i_WritePreset := stMixerAir_Valve_Int.bWritePreset,
    q_InterlocksOK => stMixerAir_Valve_Int.bInterlocksOK,
    q_TotalCycles => stMixerAir_Valve_Int.iTotalCycles,
    q_MaintCycles => stMixerAir_Valve_Int.iMaintCycles,
    q_MaintenanceCall => stMixerAir_Valve_Int.bMaintCall,
    q_State => stMixerAir_Valve_Int.iState); // FB_ValveCtrl32
stMixerAir_Valve_Int.bCmdOutWP := fbMixerAir_Valve.q_Cmd;

// NETWORK 3
OUT.bMixer_Air_V807_4 := fbMixerAir_Valve.q_Cmd;

// NETWORK 4
stMixerAir_Valve_Int.arrInterlocks := F_ToArrInterlocks(In1 := NOT OUT.bMixer_WIP_V807_3, In2 := TRUE, In3 := TRUE, In4 := TRUE, In5 := TRUE, In6 := TRUE, In7 := TRUE, In8 := TRUE);

// NETWORK 5
stMixerAir_Valve_Int.arrAlarms := F_ToArrAlarms(In1 := fbMixerAir_Valve.q_TimeoutHP, In2 := fbMixerAir_Valve.q_TimeoutWP, In3 := fbMixerAir_Valve.q_SensorsFlt, In4 := FALSE, In5 := FALSE, In6 := FALSE, In7 := FALSE, In8 := FALSE, AlarmsNOK => stMixerAir_Valve_Int.bFault);

// NETWORK 6
stMixerAir_Valve_Int.bCmdWP R= NOT stMixerAir_Valve_Int.bServiceMode;

// NETWORK 7
END_ACTION

ACTION PROD_Vacuum:
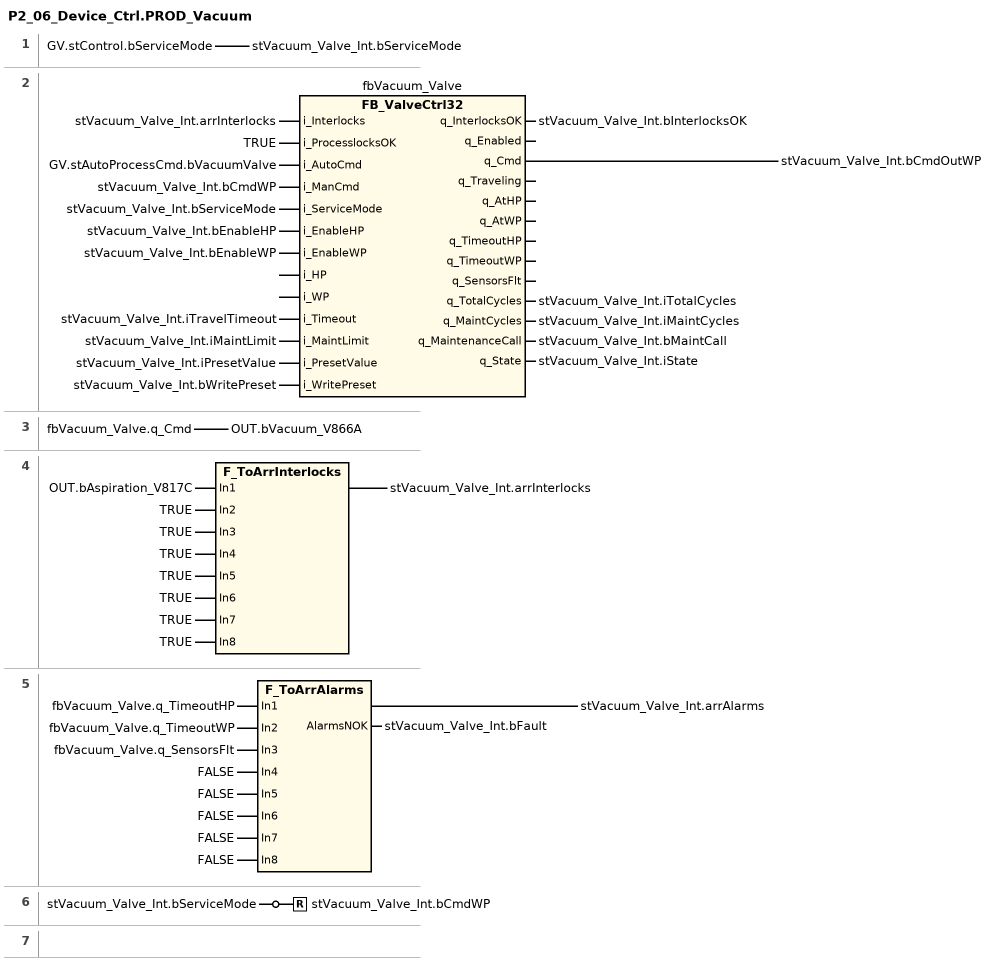
// NETWORK 1
stVacuum_Valve_Int.bServiceMode := GV.stControl.bServiceMode;

// NETWORK 2
fbVacuum_Valve(
    i_Interlocks := stVacuum_Valve_Int.arrInterlocks,
    i_ProcesslocksOK := TRUE,
    i_AutoCmd := GV.stAutoProcessCmd.bVacuumValve,
    i_ManCmd := stVacuum_Valve_Int.bCmdWP,
    i_ServiceMode := stVacuum_Valve_Int.bServiceMode,
    i_EnableHP := stVacuum_Valve_Int.bEnableHP,
    i_EnableWP := stVacuum_Valve_Int.bEnableWP,
    i_Timeout := stVacuum_Valve_Int.iTravelTimeout,
    i_MaintLimit := stVacuum_Valve_Int.iMaintLimit,
    i_PresetValue := stVacuum_Valve_Int.iPresetValue,
    i_WritePreset := stVacuum_Valve_Int.bWritePreset,
    q_InterlocksOK => stVacuum_Valve_Int.bInterlocksOK,
    q_TotalCycles => stVacuum_Valve_Int.iTotalCycles,
    q_MaintCycles => stVacuum_Valve_Int.iMaintCycles,
    q_MaintenanceCall => stVacuum_Valve_Int.bMaintCall,
    q_State => stVacuum_Valve_Int.iState); // FB_ValveCtrl32
stVacuum_Valve_Int.bCmdOutWP := fbVacuum_Valve.q_Cmd;

// NETWORK 3
OUT.bVacuum_V866A := fbVacuum_Valve.q_Cmd;

// NETWORK 4
stVacuum_Valve_Int.arrInterlocks := F_ToArrInterlocks(In1 := OUT.bAspiration_V817C, In2 := TRUE, In3 := TRUE, In4 := TRUE, In5 := TRUE, In6 := TRUE, In7 := TRUE, In8 := TRUE);

// NETWORK 5
stVacuum_Valve_Int.arrAlarms := F_ToArrAlarms(In1 := fbVacuum_Valve.q_TimeoutHP, In2 := fbVacuum_Valve.q_TimeoutWP, In3 := fbVacuum_Valve.q_SensorsFlt, In4 := FALSE, In5 := FALSE, In6 := FALSE, In7 := FALSE, In8 := FALSE, AlarmsNOK => stVacuum_Valve_Int.bFault);

// NETWORK 6
stVacuum_Valve_Int.bCmdWP R= NOT stVacuum_Valve_Int.bServiceMode;

// NETWORK 7
END_ACTION

ACTION Pump:
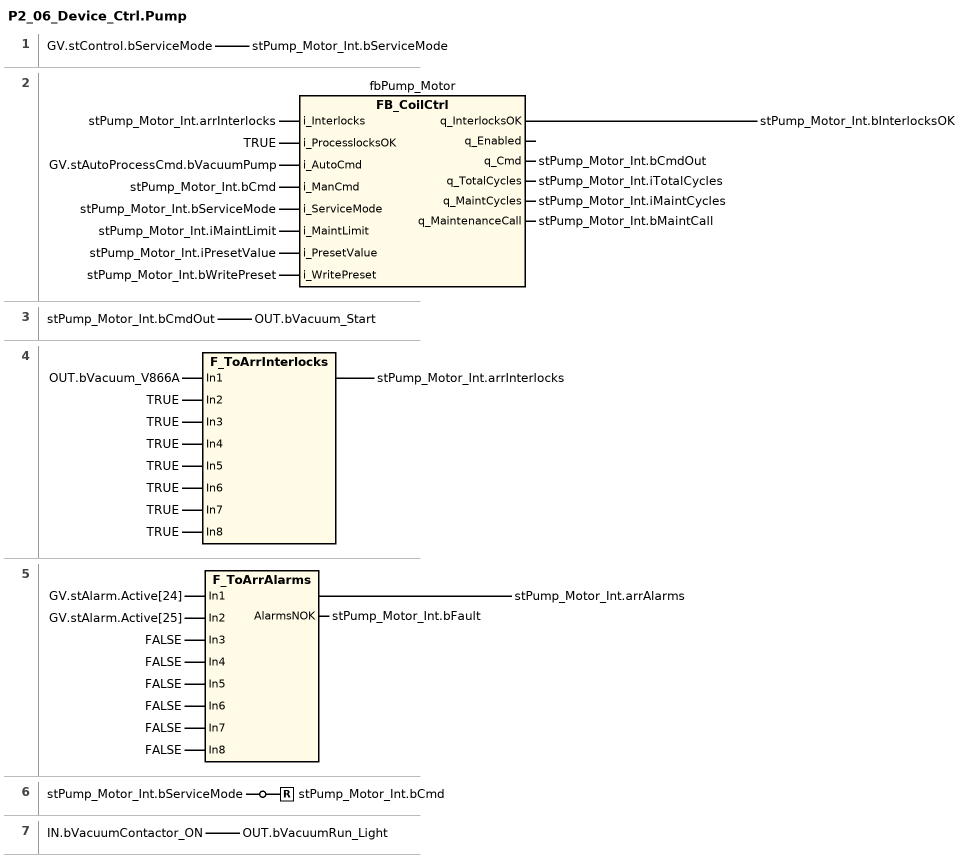
// NETWORK 1
stPump_Motor_Int.bServiceMode := GV.stControl.bServiceMode;

// NETWORK 2
fbPump_Motor(
    i_Interlocks := stPump_Motor_Int.arrInterlocks,
    i_ProcesslocksOK := TRUE,
    i_AutoCmd := GV.stAutoProcessCmd.bVacuumPump,
    i_ManCmd := stPump_Motor_Int.bCmd,
    i_ServiceMode := stPump_Motor_Int.bServiceMode,
    i_MaintLimit := stPump_Motor_Int.iMaintLimit,
    i_PresetValue := stPump_Motor_Int.iPresetValue,
    i_WritePreset := stPump_Motor_Int.bWritePreset,
    q_Cmd => stPump_Motor_Int.bCmdOut,
    q_TotalCycles => stPump_Motor_Int.iTotalCycles,
    q_MaintCycles => stPump_Motor_Int.iMaintCycles,
    q_MaintenanceCall => stPump_Motor_Int.bMaintCall); // FB_CoilCtrl
stPump_Motor_Int.bInterlocksOK := fbPump_Motor.q_InterlocksOK;

// NETWORK 3
OUT.bVacuum_Start := stPump_Motor_Int.bCmdOut;

// NETWORK 4
stPump_Motor_Int.arrInterlocks := F_ToArrInterlocks(In1 := OUT.bVacuum_V866A, In2 := TRUE, In3 := TRUE, In4 := TRUE, In5 := TRUE, In6 := TRUE, In7 := TRUE, In8 := TRUE);

// NETWORK 5
stPump_Motor_Int.arrAlarms := F_ToArrAlarms(In1 := GV.stAlarm.Active[24], In2 := GV.stAlarm.Active[25], In3 := FALSE, In4 := FALSE, In5 := FALSE, In6 := FALSE, In7 := FALSE, In8 := FALSE, AlarmsNOK => stPump_Motor_Int.bFault);

// NETWORK 6
stPump_Motor_Int.bCmd R= NOT stPump_Motor_Int.bServiceMode;

// NETWORK 7
OUT.bVacuumRun_Light := IN.bVacuumContactor_ON;
END_ACTION

ACTION Purge:
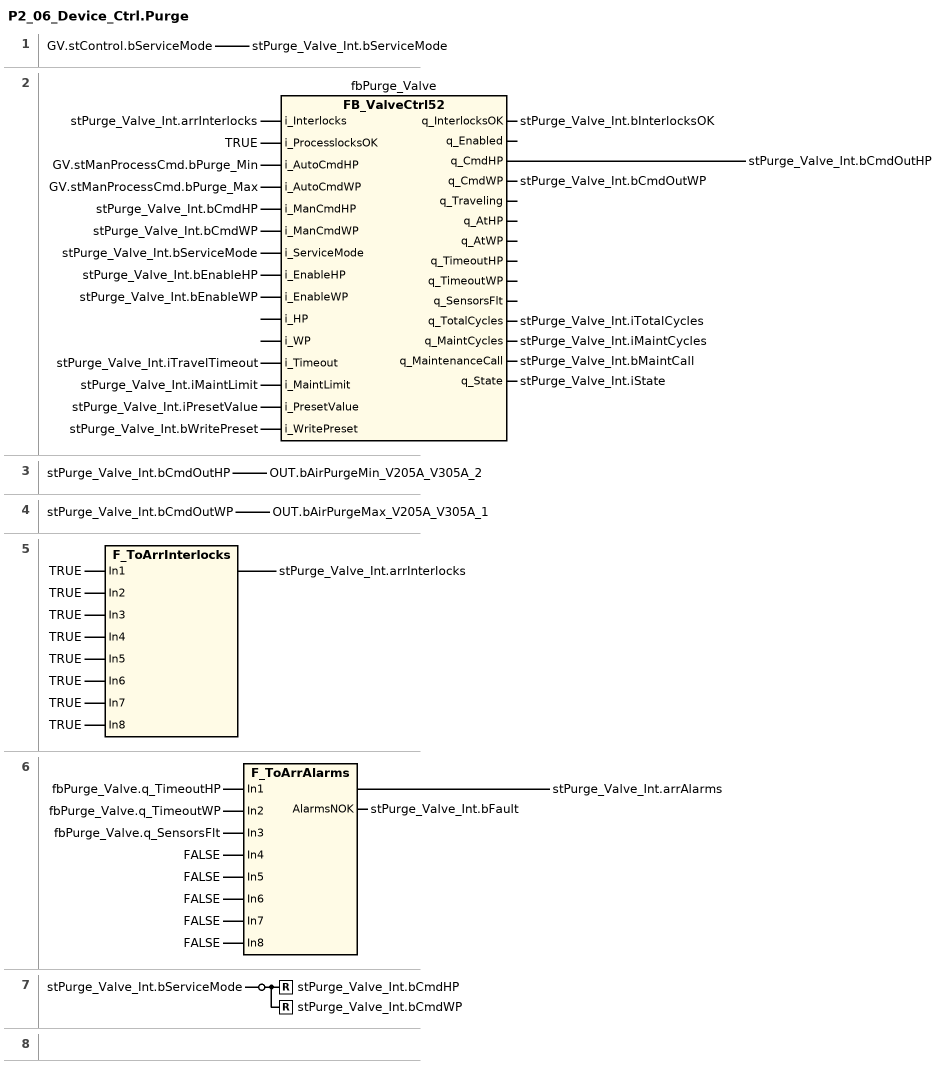
// NETWORK 1
stPurge_Valve_Int.bServiceMode := GV.stControl.bServiceMode;

// NETWORK 2
fbPurge_Valve(
    i_Interlocks := stPurge_Valve_Int.arrInterlocks,
    i_ProcesslocksOK := TRUE,
    i_AutoCmdHP := GV.stManProcessCmd.bPurge_Min,
    i_AutoCmdWP := GV.stManProcessCmd.bPurge_Max,
    i_ManCmdHP := stPurge_Valve_Int.bCmdHP,
    i_ManCmdWP := stPurge_Valve_Int.bCmdWP,
    i_ServiceMode := stPurge_Valve_Int.bServiceMode,
    i_EnableHP := stPurge_Valve_Int.bEnableHP,
    i_EnableWP := stPurge_Valve_Int.bEnableWP,
    i_Timeout := stPurge_Valve_Int.iTravelTimeout,
    i_MaintLimit := stPurge_Valve_Int.iMaintLimit,
    i_PresetValue := stPurge_Valve_Int.iPresetValue,
    i_WritePreset := stPurge_Valve_Int.bWritePreset,
    q_InterlocksOK => stPurge_Valve_Int.bInterlocksOK,
    q_CmdWP => stPurge_Valve_Int.bCmdOutWP,
    q_TotalCycles => stPurge_Valve_Int.iTotalCycles,
    q_MaintCycles => stPurge_Valve_Int.iMaintCycles,
    q_MaintenanceCall => stPurge_Valve_Int.bMaintCall,
    q_State => stPurge_Valve_Int.iState); // FB_ValveCtrl52
stPurge_Valve_Int.bCmdOutHP := fbPurge_Valve.q_CmdHP;

// NETWORK 3
OUT.bAirPurgeMin_V205A_V305A_2 := stPurge_Valve_Int.bCmdOutHP;

// NETWORK 4
OUT.bAirPurgeMax_V205A_V305A_1 := stPurge_Valve_Int.bCmdOutWP;

// NETWORK 5
stPurge_Valve_Int.arrInterlocks := F_ToArrInterlocks(In1 := TRUE, In2 := TRUE, In3 := TRUE, In4 := TRUE, In5 := TRUE, In6 := TRUE, In7 := TRUE, In8 := TRUE);

// NETWORK 6
stPurge_Valve_Int.arrAlarms := F_ToArrAlarms(In1 := fbPurge_Valve.q_TimeoutHP, In2 := fbPurge_Valve.q_TimeoutWP, In3 := fbPurge_Valve.q_SensorsFlt, In4 := FALSE, In5 := FALSE, In6 := FALSE, In7 := FALSE, In8 := FALSE, AlarmsNOK => stPurge_Valve_Int.bFault);

// NETWORK 7
_w5 := NOT stPurge_Valve_Int.bServiceMode;
stPurge_Valve_Int.bCmdHP R= _w5;
stPurge_Valve_Int.bCmdWP R= _w5;

// NETWORK 8
END_ACTION

ACTION Seal:
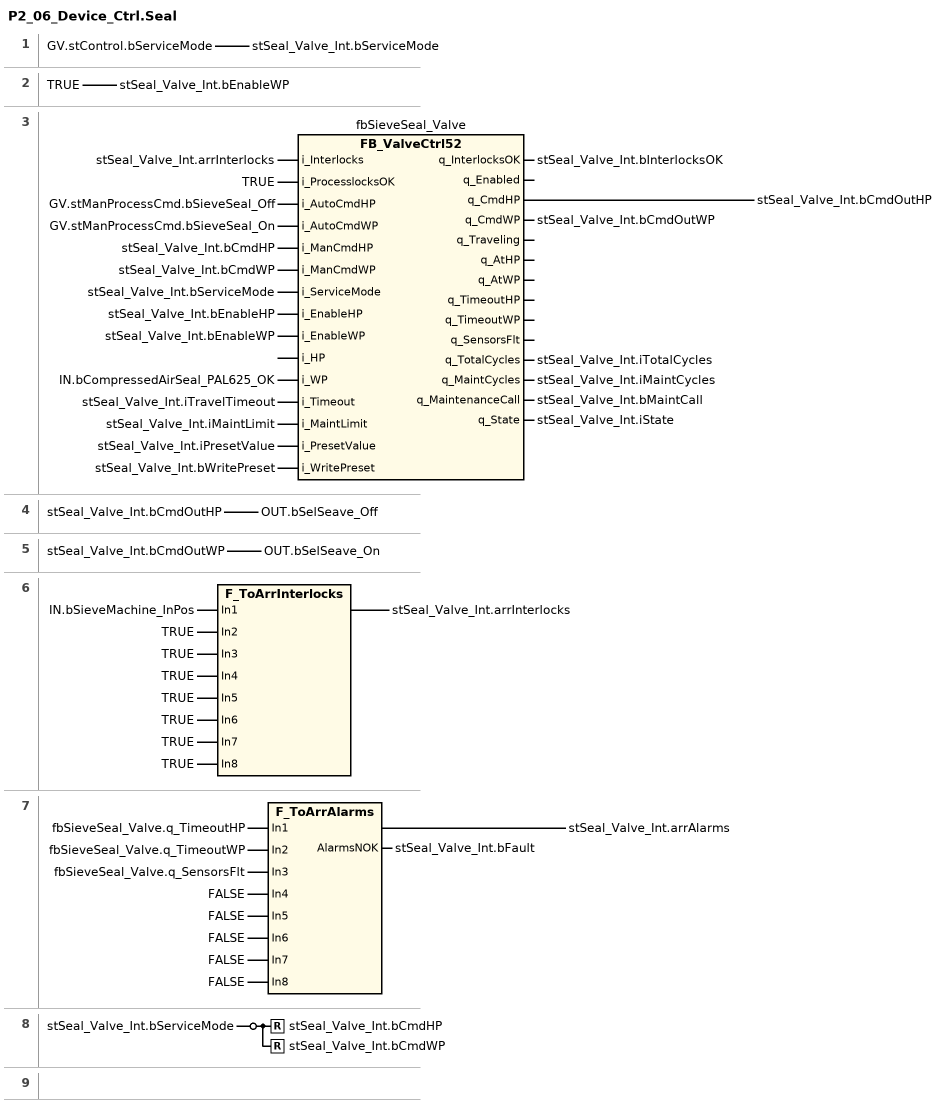
// NETWORK 1
stSeal_Valve_Int.bServiceMode := GV.stControl.bServiceMode;

// NETWORK 2
stSeal_Valve_Int.bEnableWP := TRUE;

// NETWORK 3
fbSieveSeal_Valve(
    i_Interlocks := stSeal_Valve_Int.arrInterlocks,
    i_ProcesslocksOK := TRUE,
    i_AutoCmdHP := GV.stManProcessCmd.bSieveSeal_Off,
    i_AutoCmdWP := GV.stManProcessCmd.bSieveSeal_On,
    i_ManCmdHP := stSeal_Valve_Int.bCmdHP,
    i_ManCmdWP := stSeal_Valve_Int.bCmdWP,
    i_ServiceMode := stSeal_Valve_Int.bServiceMode,
    i_EnableHP := stSeal_Valve_Int.bEnableHP,
    i_EnableWP := stSeal_Valve_Int.bEnableWP,
    i_WP := IN.bCompressedAirSeal_PAL625_OK,
    i_Timeout := stSeal_Valve_Int.iTravelTimeout,
    i_MaintLimit := stSeal_Valve_Int.iMaintLimit,
    i_PresetValue := stSeal_Valve_Int.iPresetValue,
    i_WritePreset := stSeal_Valve_Int.bWritePreset,
    q_InterlocksOK => stSeal_Valve_Int.bInterlocksOK,
    q_CmdWP => stSeal_Valve_Int.bCmdOutWP,
    q_TotalCycles => stSeal_Valve_Int.iTotalCycles,
    q_MaintCycles => stSeal_Valve_Int.iMaintCycles,
    q_MaintenanceCall => stSeal_Valve_Int.bMaintCall,
    q_State => stSeal_Valve_Int.iState); // FB_ValveCtrl52
stSeal_Valve_Int.bCmdOutHP := fbSieveSeal_Valve.q_CmdHP;

// NETWORK 4
OUT.bSelSeave_Off := stSeal_Valve_Int.bCmdOutHP;

// NETWORK 5
OUT.bSelSeave_On := stSeal_Valve_Int.bCmdOutWP;

// NETWORK 6
stSeal_Valve_Int.arrInterlocks := F_ToArrInterlocks(In1 := IN.bSieveMachine_InPos, In2 := TRUE, In3 := TRUE, In4 := TRUE, In5 := TRUE, In6 := TRUE, In7 := TRUE, In8 := TRUE);

// NETWORK 7
stSeal_Valve_Int.arrAlarms := F_ToArrAlarms(In1 := fbSieveSeal_Valve.q_TimeoutHP, In2 := fbSieveSeal_Valve.q_TimeoutWP, In3 := fbSieveSeal_Valve.q_SensorsFlt, In4 := FALSE, In5 := FALSE, In6 := FALSE, In7 := FALSE, In8 := FALSE, AlarmsNOK => stSeal_Valve_Int.bFault);

// NETWORK 8
_w6 := NOT stSeal_Valve_Int.bServiceMode;
stSeal_Valve_Int.bCmdHP R= _w6;
stSeal_Valve_Int.bCmdWP R= _w6;

// NETWORK 9
END_ACTION

ACTION Sieve:
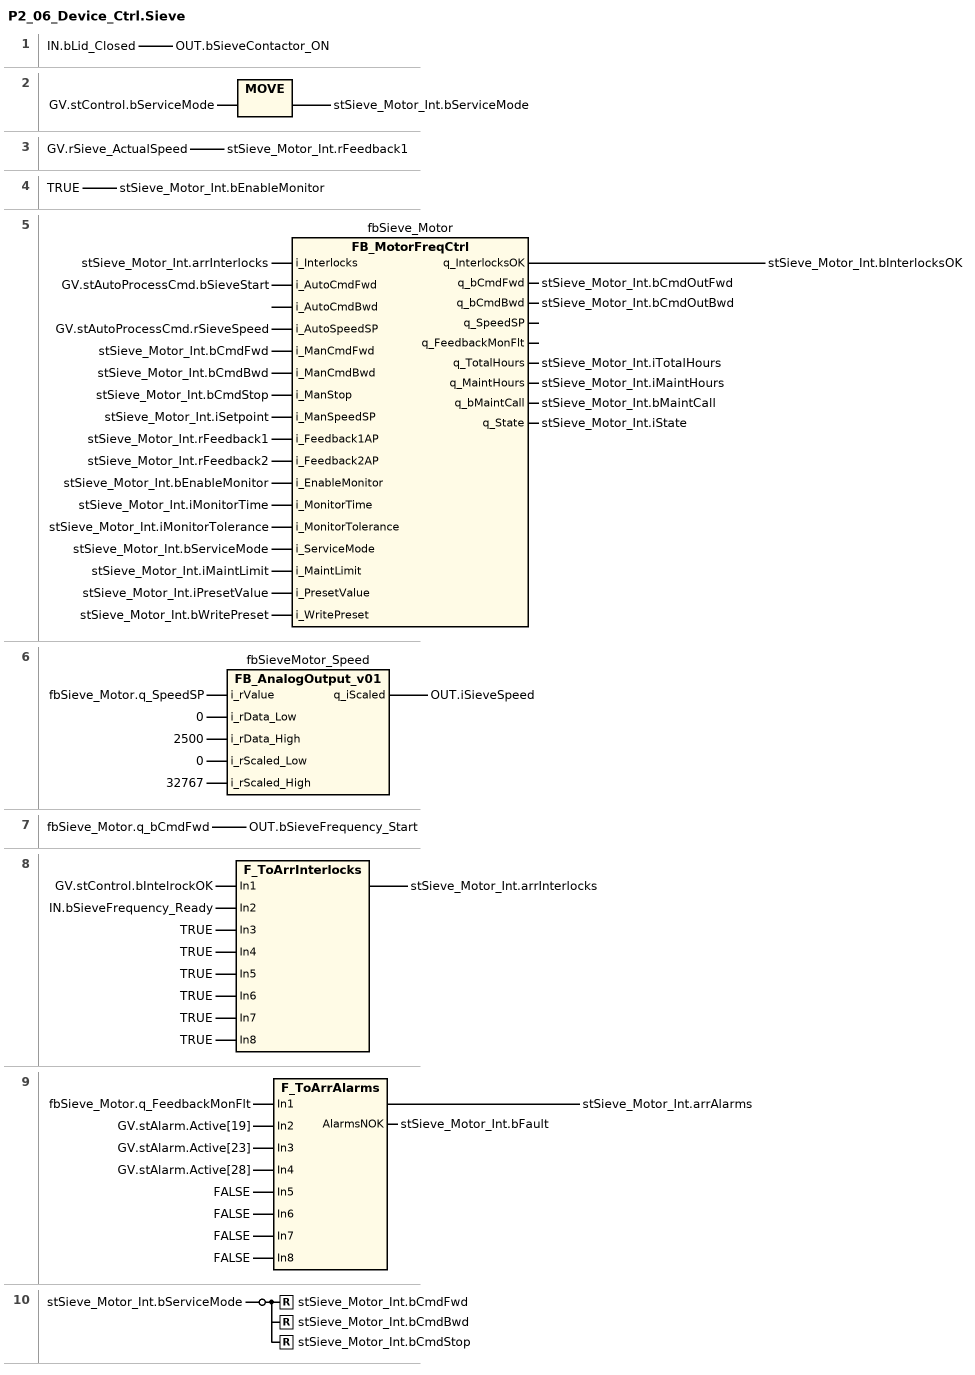
// NETWORK 1
OUT.bSieveContactor_ON := IN.bLid_Closed;

// NETWORK 2
stSieve_Motor_Int.bServiceMode := GV.stControl.bServiceMode;

// NETWORK 3
stSieve_Motor_Int.rFeedback1 := GV.rSieve_ActualSpeed;

// NETWORK 4
stSieve_Motor_Int.bEnableMonitor := TRUE;

// NETWORK 5
fbSieve_Motor(
    i_Interlocks := stSieve_Motor_Int.arrInterlocks,
    i_AutoCmdFwd := GV.stAutoProcessCmd.bSieveStart,
    i_AutoSpeedSP := GV.stAutoProcessCmd.rSieveSpeed,
    i_ManCmdFwd := stSieve_Motor_Int.bCmdFwd,
    i_ManCmdBwd := stSieve_Motor_Int.bCmdBwd,
    i_ManStop := stSieve_Motor_Int.bCmdStop,
    i_ManSpeedSP := stSieve_Motor_Int.iSetpoint,
    i_Feedback1AP := stSieve_Motor_Int.rFeedback1,
    i_Feedback2AP := stSieve_Motor_Int.rFeedback2,
    i_EnableMonitor := stSieve_Motor_Int.bEnableMonitor,
    i_MonitorTime := stSieve_Motor_Int.iMonitorTime,
    i_MonitorTolerance := stSieve_Motor_Int.iMonitorTolerance,
    i_ServiceMode := stSieve_Motor_Int.bServiceMode,
    i_MaintLimit := stSieve_Motor_Int.iMaintLimit,
    i_PresetValue := stSieve_Motor_Int.iPresetValue,
    i_WritePreset := stSieve_Motor_Int.bWritePreset,
    q_bCmdFwd => stSieve_Motor_Int.bCmdOutFwd,
    q_bCmdBwd => stSieve_Motor_Int.bCmdOutBwd,
    q_TotalHours => stSieve_Motor_Int.iTotalHours,
    q_MaintHours => stSieve_Motor_Int.iMaintHours,
    q_bMaintCall => stSieve_Motor_Int.bMaintCall,
    q_State => stSieve_Motor_Int.iState); // FB_MotorFreqCtrl
stSieve_Motor_Int.bInterlocksOK := fbSieve_Motor.q_InterlocksOK;

// NETWORK 6
fbSieveMotor_Speed(
    i_rValue := fbSieve_Motor.q_SpeedSP,
    i_rData_Low := 0,
    i_rData_High := 2500,
    i_rScaled_Low := 0,
    i_rScaled_High := 32767); // FB_AnalogOutput_v01
OUT.iSieveSpeed := fbSieveMotor_Speed.q_iScaled;

// NETWORK 7
OUT.bSieveFrequency_Start := fbSieve_Motor.q_bCmdFwd;

// NETWORK 8
stSieve_Motor_Int.arrInterlocks := F_ToArrInterlocks(In1 := GV.stControl.bIntelrockOK, In2 := IN.bSieveFrequency_Ready, In3 := TRUE, In4 := TRUE, In5 := TRUE, In6 := TRUE, In7 := TRUE, In8 := TRUE);

// NETWORK 9
stSieve_Motor_Int.arrAlarms := F_ToArrAlarms(In1 := fbSieve_Motor.q_FeedbackMonFlt, In2 := GV.stAlarm.Active[19], In3 := GV.stAlarm.Active[23], In4 := GV.stAlarm.Active[28], In5 := FALSE, In6 := FALSE, In7 := FALSE, In8 := FALSE, AlarmsNOK => stSieve_Motor_Int.bFault);

// NETWORK 10
_w7 := NOT stSieve_Motor_Int.bServiceMode;
stSieve_Motor_Int.bCmdFwd R= _w7;
stSieve_Motor_Int.bCmdBwd R= _w7;
stSieve_Motor_Int.bCmdStop R= _w7;

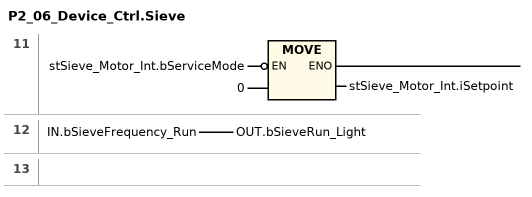
// NETWORK 11
IF NOT stSieve_Motor_Int.bServiceMode THEN stSieve_Motor_Int.iSetpoint := 0; END_IF

// NETWORK 12
OUT.bSieveRun_Light := IN.bSieveFrequency_Run;

// NETWORK 13
END_ACTION

ACTION SP_Mixer:
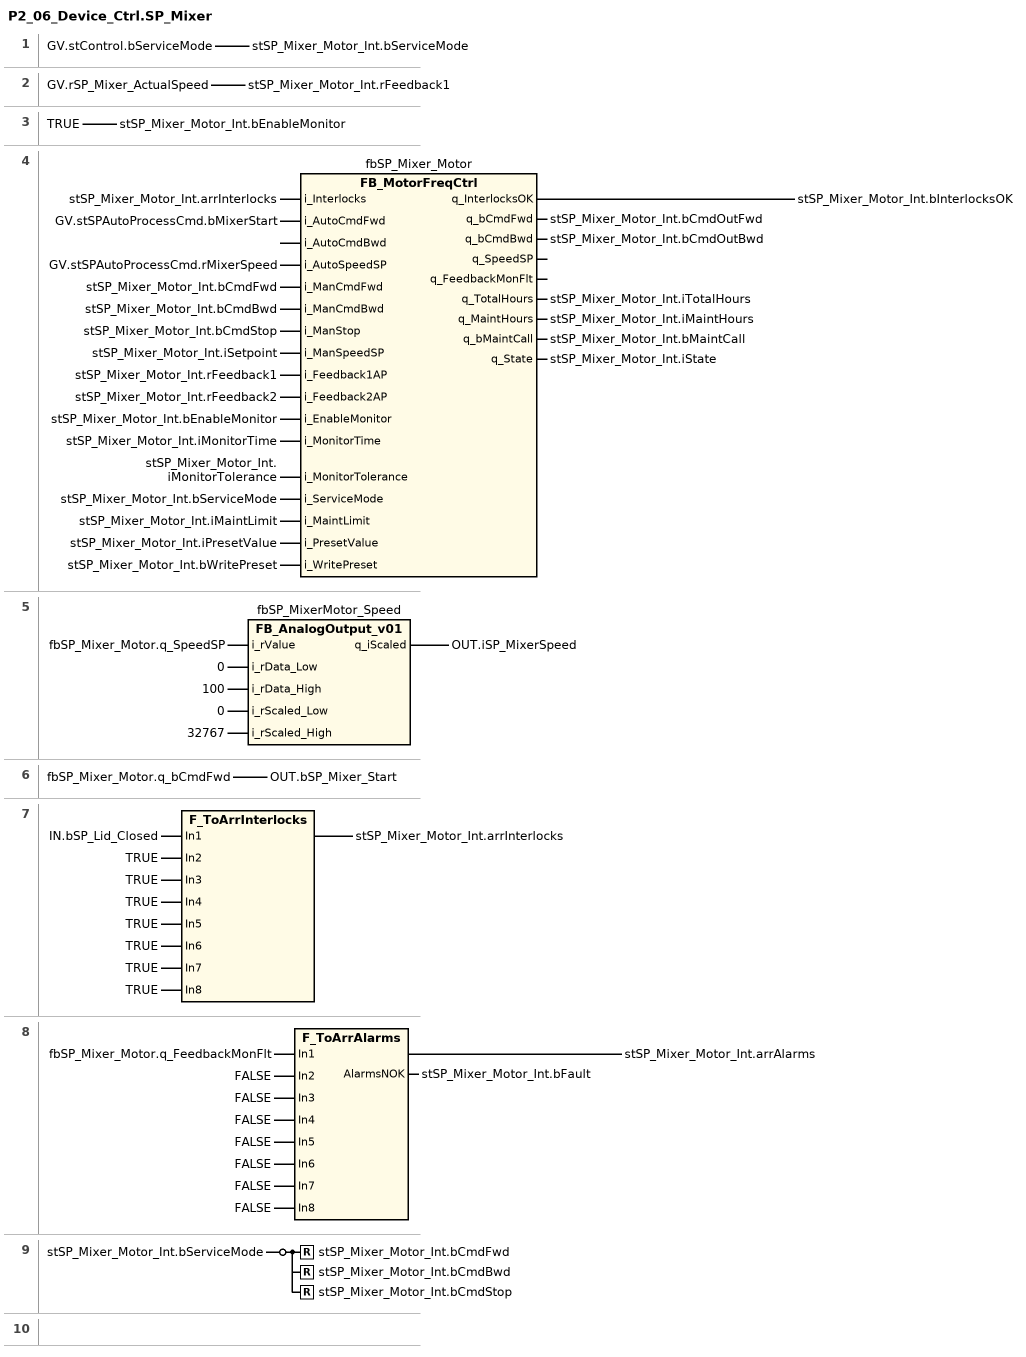
// NETWORK 1
stSP_Mixer_Motor_Int.bServiceMode := GV.stControl.bServiceMode;

// NETWORK 2
stSP_Mixer_Motor_Int.rFeedback1 := GV.rSP_Mixer_ActualSpeed;

// NETWORK 3
stSP_Mixer_Motor_Int.bEnableMonitor := TRUE;

// NETWORK 4
fbSP_Mixer_Motor(
    i_Interlocks := stSP_Mixer_Motor_Int.arrInterlocks,
    i_AutoCmdFwd := GV.stSPAutoProcessCmd.bMixerStart,
    i_AutoSpeedSP := GV.stSPAutoProcessCmd.rMixerSpeed,
    i_ManCmdFwd := stSP_Mixer_Motor_Int.bCmdFwd,
    i_ManCmdBwd := stSP_Mixer_Motor_Int.bCmdBwd,
    i_ManStop := stSP_Mixer_Motor_Int.bCmdStop,
    i_ManSpeedSP := stSP_Mixer_Motor_Int.iSetpoint,
    i_Feedback1AP := stSP_Mixer_Motor_Int.rFeedback1,
    i_Feedback2AP := stSP_Mixer_Motor_Int.rFeedback2,
    i_EnableMonitor := stSP_Mixer_Motor_Int.bEnableMonitor,
    i_MonitorTime := stSP_Mixer_Motor_Int.iMonitorTime,
    i_MonitorTolerance := stSP_Mixer_Motor_Int.iMonitorTolerance,
    i_ServiceMode := stSP_Mixer_Motor_Int.bServiceMode,
    i_MaintLimit := stSP_Mixer_Motor_Int.iMaintLimit,
    i_PresetValue := stSP_Mixer_Motor_Int.iPresetValue,
    i_WritePreset := stSP_Mixer_Motor_Int.bWritePreset,
    q_bCmdFwd => stSP_Mixer_Motor_Int.bCmdOutFwd,
    q_bCmdBwd => stSP_Mixer_Motor_Int.bCmdOutBwd,
    q_TotalHours => stSP_Mixer_Motor_Int.iTotalHours,
    q_MaintHours => stSP_Mixer_Motor_Int.iMaintHours,
    q_bMaintCall => stSP_Mixer_Motor_Int.bMaintCall,
    q_State => stSP_Mixer_Motor_Int.iState); // FB_MotorFreqCtrl
stSP_Mixer_Motor_Int.bInterlocksOK := fbSP_Mixer_Motor.q_InterlocksOK;

// NETWORK 5
fbSP_MixerMotor_Speed(
    i_rValue := fbSP_Mixer_Motor.q_SpeedSP,
    i_rData_Low := 0,
    i_rData_High := 100,
    i_rScaled_Low := 0,
    i_rScaled_High := 32767); // FB_AnalogOutput_v01
OUT.iSP_MixerSpeed := fbSP_MixerMotor_Speed.q_iScaled;

// NETWORK 6
OUT.bSP_Mixer_Start := fbSP_Mixer_Motor.q_bCmdFwd;

// NETWORK 7
stSP_Mixer_Motor_Int.arrInterlocks := F_ToArrInterlocks(In1 := IN.bSP_Lid_Closed, In2 := TRUE, In3 := TRUE, In4 := TRUE, In5 := TRUE, In6 := TRUE, In7 := TRUE, In8 := TRUE);

// NETWORK 8
stSP_Mixer_Motor_Int.arrAlarms := F_ToArrAlarms(In1 := fbSP_Mixer_Motor.q_FeedbackMonFlt, In2 := FALSE, In3 := FALSE, In4 := FALSE, In5 := FALSE, In6 := FALSE, In7 := FALSE, In8 := FALSE, AlarmsNOK => stSP_Mixer_Motor_Int.bFault);

// NETWORK 9
_w8 := NOT stSP_Mixer_Motor_Int.bServiceMode;
stSP_Mixer_Motor_Int.bCmdFwd R= _w8;
stSP_Mixer_Motor_Int.bCmdBwd R= _w8;
stSP_Mixer_Motor_Int.bCmdStop R= _w8;

// NETWORK 10
END_ACTION

ACTION SP_Pressure:
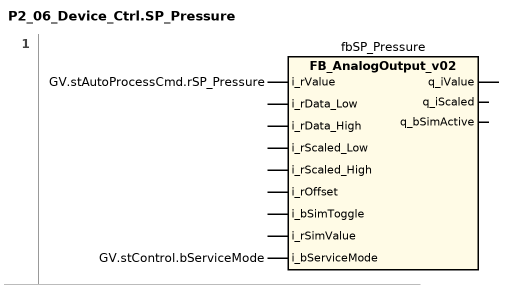
// NETWORK 1
fbSP_Pressure(i_rValue := GV.stAutoProcessCmd.rSP_Pressure, i_bServiceMode := GV.stControl.bServiceMode); // FB_AnalogOutput_v02
END_ACTION

ACTION SP_Temperature:
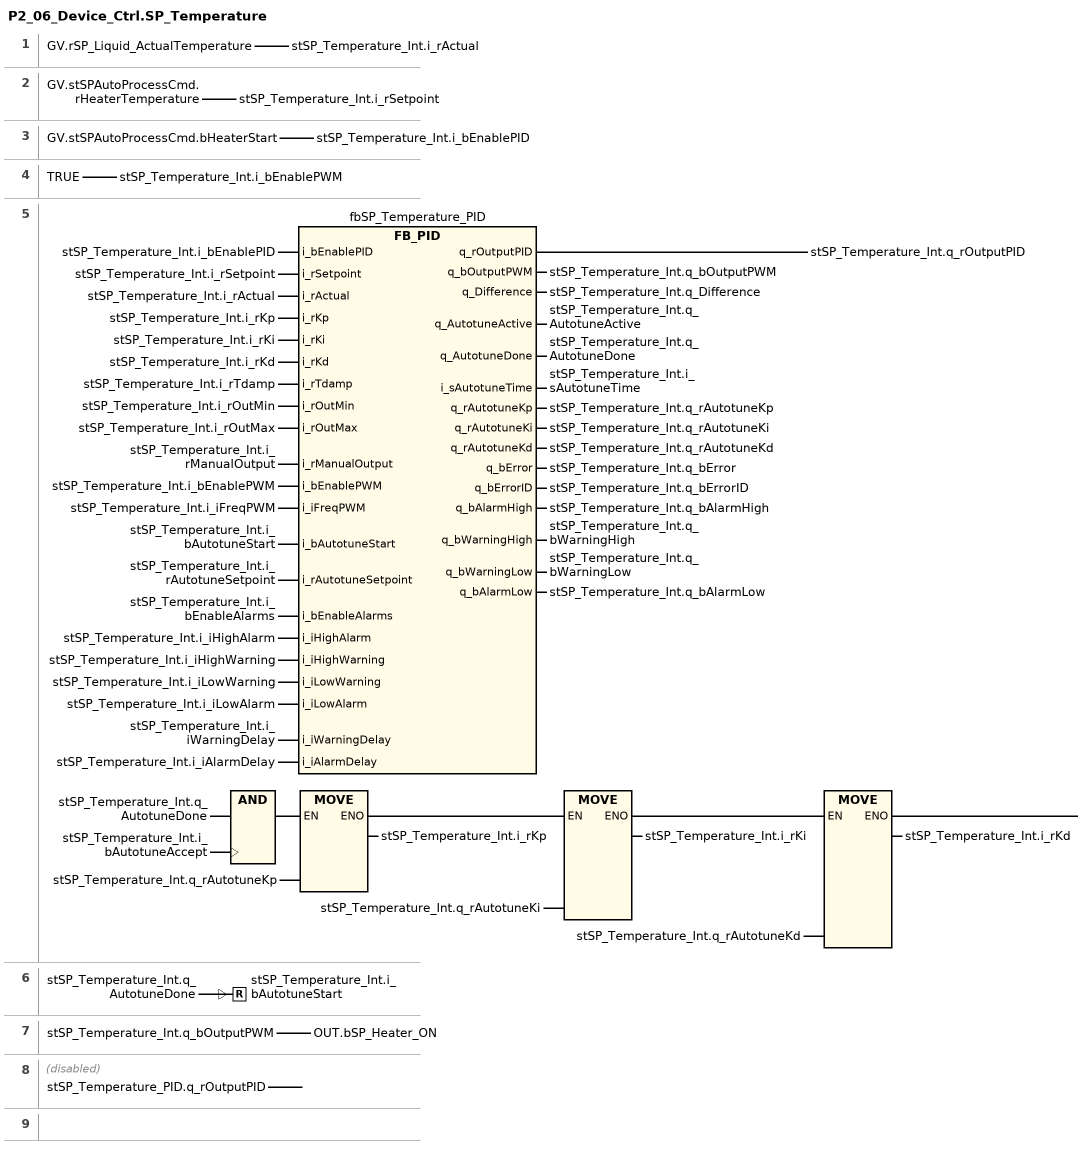
// NETWORK 1
stSP_Temperature_Int.i_rActual := GV.rSP_Liquid_ActualTemperature;

// NETWORK 2
stSP_Temperature_Int.i_rSetpoint := GV.stSPAutoProcessCmd.rHeaterTemperature;

// NETWORK 3
stSP_Temperature_Int.i_bEnablePID := GV.stSPAutoProcessCmd.bHeaterStart;

// NETWORK 4
stSP_Temperature_Int.i_bEnablePWM := TRUE;

// NETWORK 5
fbSP_Temperature_PID(
    i_bEnablePID := stSP_Temperature_Int.i_bEnablePID,
    i_rSetpoint := stSP_Temperature_Int.i_rSetpoint,
    i_rActual := stSP_Temperature_Int.i_rActual,
    i_rKp := stSP_Temperature_Int.i_rKp,
    i_rKi := stSP_Temperature_Int.i_rKi,
    i_rKd := stSP_Temperature_Int.i_rKd,
    i_rTdamp := stSP_Temperature_Int.i_rTdamp,
    i_rOutMin := stSP_Temperature_Int.i_rOutMin,
    i_rOutMax := stSP_Temperature_Int.i_rOutMax,
    i_rManualOutput := stSP_Temperature_Int.i_rManualOutput,
    i_bEnablePWM := stSP_Temperature_Int.i_bEnablePWM,
    i_iFreqPWM := stSP_Temperature_Int.i_iFreqPWM,
    i_bAutotuneStart := stSP_Temperature_Int.i_bAutotuneStart,
    i_rAutotuneSetpoint := stSP_Temperature_Int.i_rAutotuneSetpoint,
    i_bEnableAlarms := stSP_Temperature_Int.i_bEnableAlarms,
    i_iHighAlarm := stSP_Temperature_Int.i_iHighAlarm,
    i_iHighWarning := stSP_Temperature_Int.i_iHighWarning,
    i_iLowWarning := stSP_Temperature_Int.i_iLowWarning,
    i_iLowAlarm := stSP_Temperature_Int.i_iLowAlarm,
    i_iWarningDelay := stSP_Temperature_Int.i_iWarningDelay,
    i_iAlarmDelay := stSP_Temperature_Int.i_iAlarmDelay,
    q_bOutputPWM => stSP_Temperature_Int.q_bOutputPWM,
    q_Difference => stSP_Temperature_Int.q_Difference,
    q_AutotuneActive => stSP_Temperature_Int.q_AutotuneActive,
    q_AutotuneDone => stSP_Temperature_Int.q_AutotuneDone,
    i_sAutotuneTime => stSP_Temperature_Int.i_sAutotuneTime,
    q_rAutotuneKp => stSP_Temperature_Int.q_rAutotuneKp,
    q_rAutotuneKi => stSP_Temperature_Int.q_rAutotuneKi,
    q_rAutotuneKd => stSP_Temperature_Int.q_rAutotuneKd,
    q_bError => stSP_Temperature_Int.q_bError,
    q_bErrorID => stSP_Temperature_Int.q_bErrorID,
    q_bAlarmHigh => stSP_Temperature_Int.q_bAlarmHigh,
    q_bWarningHigh => stSP_Temperature_Int.q_bWarningHigh,
    q_bWarningLow => stSP_Temperature_Int.q_bWarningLow,
    q_bAlarmLow => stSP_Temperature_Int.q_bAlarmLow); // FB_PID
stSP_Temperature_Int.q_rOutputPID := fbSP_Temperature_PID.q_rOutputPID;
_rt1(CLK := stSP_Temperature_Int.i_bAutotuneAccept);
_w9 := stSP_Temperature_Int.q_AutotuneDone AND _rt1.Q;
IF _w9 THEN stSP_Temperature_Int.i_rKp := stSP_Temperature_Int.q_rAutotuneKp; END_IF
IF _w9 THEN stSP_Temperature_Int.i_rKi := stSP_Temperature_Int.q_rAutotuneKi; END_IF
IF _w9 THEN stSP_Temperature_Int.i_rKd := stSP_Temperature_Int.q_rAutotuneKd; END_IF

// NETWORK 6
_rt2(CLK := stSP_Temperature_Int.q_AutotuneDone);
stSP_Temperature_Int.i_bAutotuneStart R= _rt2.Q;

// NETWORK 7
OUT.bSP_Heater_ON := stSP_Temperature_Int.q_bOutputPWM;

// NETWORK 8 (disabled)
// ??? := stSP_Temperature_PID.q_rOutputPID;

// NETWORK 9
END_ACTION

ACTION Tool:
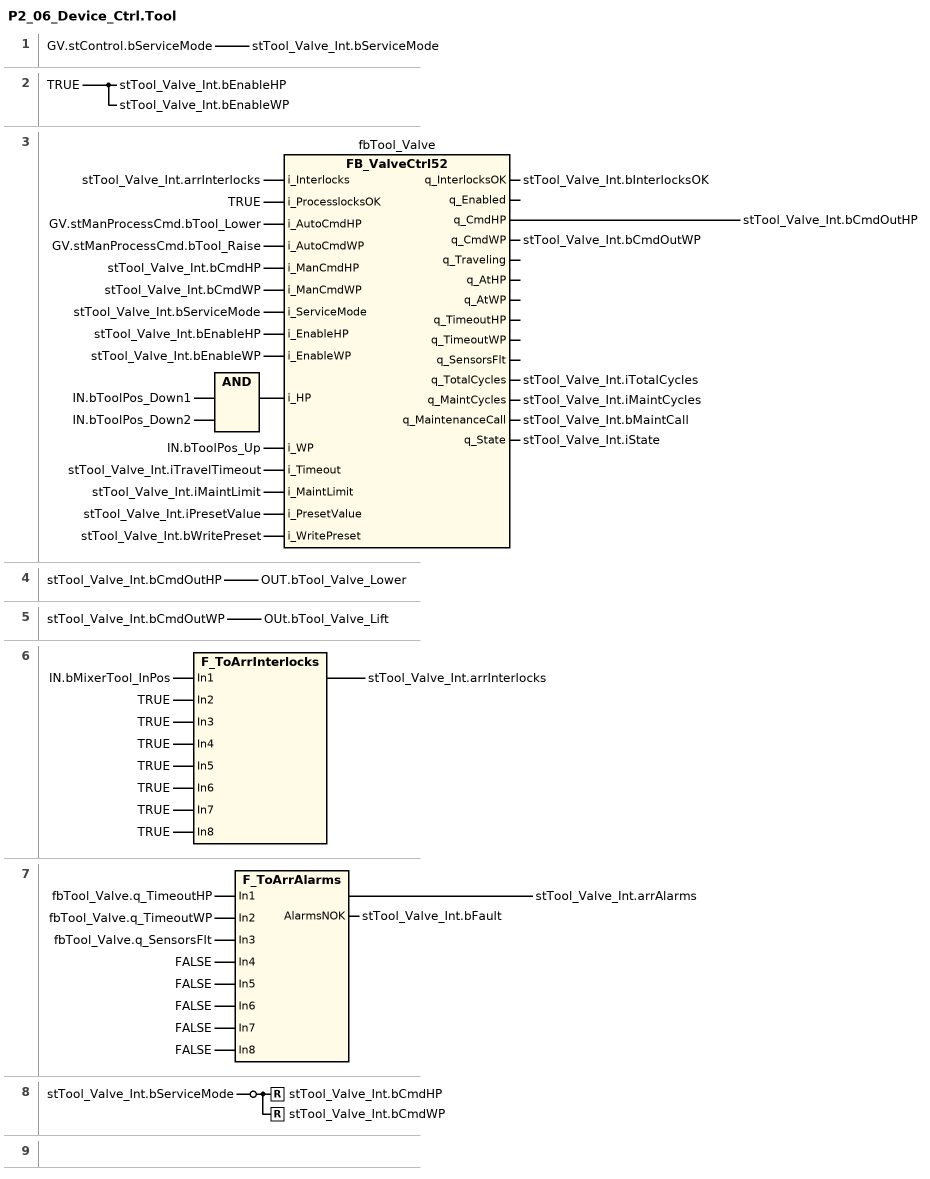
// NETWORK 1
stTool_Valve_Int.bServiceMode := GV.stControl.bServiceMode;

// NETWORK 2
stTool_Valve_Int.bEnableHP := TRUE;
stTool_Valve_Int.bEnableWP := TRUE;

// NETWORK 3
fbTool_Valve(
    i_Interlocks := stTool_Valve_Int.arrInterlocks,
    i_ProcesslocksOK := TRUE,
    i_AutoCmdHP := GV.stManProcessCmd.bTool_Lower,
    i_AutoCmdWP := GV.stManProcessCmd.bTool_Raise,
    i_ManCmdHP := stTool_Valve_Int.bCmdHP,
    i_ManCmdWP := stTool_Valve_Int.bCmdWP,
    i_ServiceMode := stTool_Valve_Int.bServiceMode,
    i_EnableHP := stTool_Valve_Int.bEnableHP,
    i_EnableWP := stTool_Valve_Int.bEnableWP,
    i_HP := IN.bToolPos_Down1 AND IN.bToolPos_Down2,
    i_WP := IN.bToolPos_Up,
    i_Timeout := stTool_Valve_Int.iTravelTimeout,
    i_MaintLimit := stTool_Valve_Int.iMaintLimit,
    i_PresetValue := stTool_Valve_Int.iPresetValue,
    i_WritePreset := stTool_Valve_Int.bWritePreset,
    q_InterlocksOK => stTool_Valve_Int.bInterlocksOK,
    q_CmdWP => stTool_Valve_Int.bCmdOutWP,
    q_TotalCycles => stTool_Valve_Int.iTotalCycles,
    q_MaintCycles => stTool_Valve_Int.iMaintCycles,
    q_MaintenanceCall => stTool_Valve_Int.bMaintCall,
    q_State => stTool_Valve_Int.iState); // FB_ValveCtrl52
stTool_Valve_Int.bCmdOutHP := fbTool_Valve.q_CmdHP;

// NETWORK 4
OUT.bTool_Valve_Lower := stTool_Valve_Int.bCmdOutHP;

// NETWORK 5
OUt.bTool_Valve_Lift := stTool_Valve_Int.bCmdOutWP;

// NETWORK 6
stTool_Valve_Int.arrInterlocks := F_ToArrInterlocks(In1 := IN.bMixerTool_InPos, In2 := TRUE, In3 := TRUE, In4 := TRUE, In5 := TRUE, In6 := TRUE, In7 := TRUE, In8 := TRUE);

// NETWORK 7
stTool_Valve_Int.arrAlarms := F_ToArrAlarms(In1 := fbTool_Valve.q_TimeoutHP, In2 := fbTool_Valve.q_TimeoutWP, In3 := fbTool_Valve.q_SensorsFlt, In4 := FALSE, In5 := FALSE, In6 := FALSE, In7 := FALSE, In8 := FALSE, AlarmsNOK => stTool_Valve_Int.bFault);

// NETWORK 8
_w10 := NOT stTool_Valve_Int.bServiceMode;
stTool_Valve_Int.bCmdHP R= _w10;
stTool_Valve_Int.bCmdWP R= _w10;

// NETWORK 9
END_ACTION

ACTION WIP_Chopper:
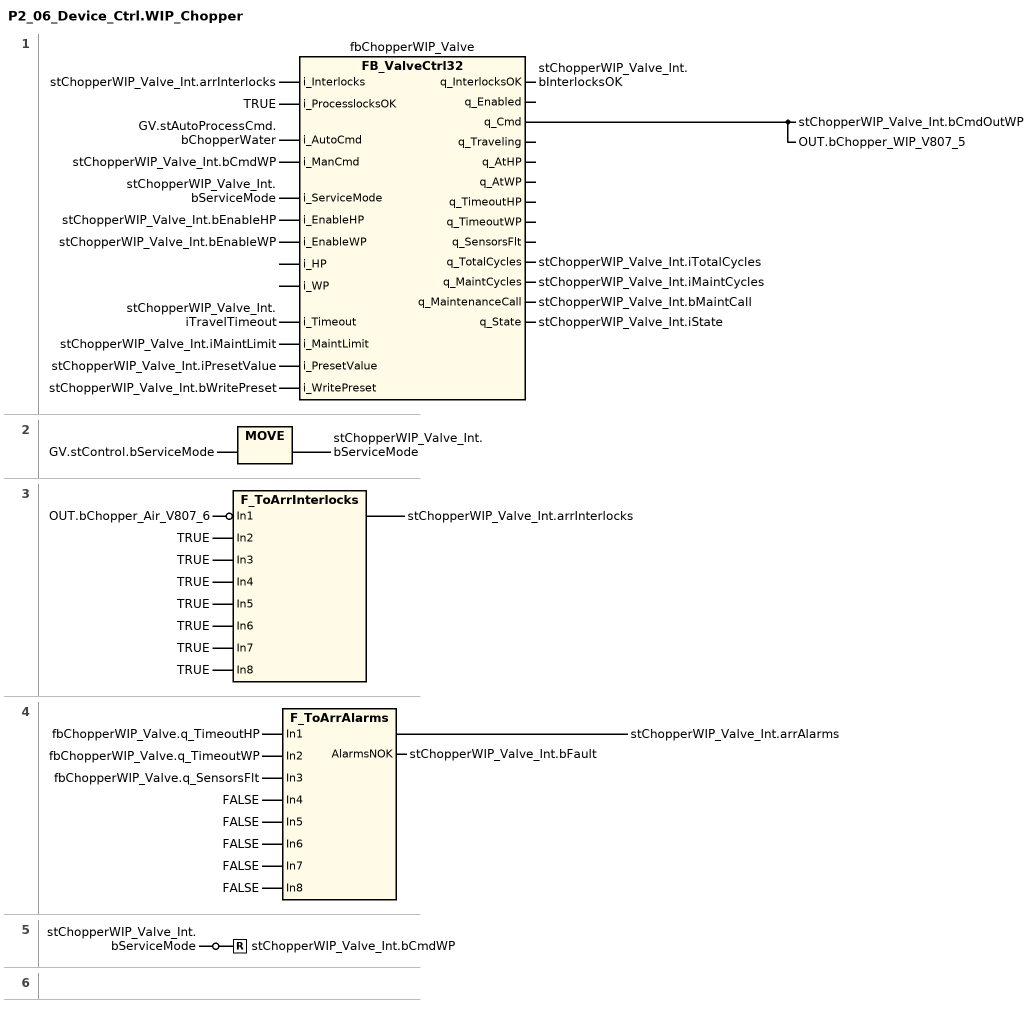
// NETWORK 1
fbChopperWIP_Valve(
    i_Interlocks := stChopperWIP_Valve_Int.arrInterlocks,
    i_ProcesslocksOK := TRUE,
    i_AutoCmd := GV.stAutoProcessCmd.bChopperWater,
    i_ManCmd := stChopperWIP_Valve_Int.bCmdWP,
    i_ServiceMode := stChopperWIP_Valve_Int.bServiceMode,
    i_EnableHP := stChopperWIP_Valve_Int.bEnableHP,
    i_EnableWP := stChopperWIP_Valve_Int.bEnableWP,
    i_Timeout := stChopperWIP_Valve_Int.iTravelTimeout,
    i_MaintLimit := stChopperWIP_Valve_Int.iMaintLimit,
    i_PresetValue := stChopperWIP_Valve_Int.iPresetValue,
    i_WritePreset := stChopperWIP_Valve_Int.bWritePreset,
    q_InterlocksOK => stChopperWIP_Valve_Int.bInterlocksOK,
    q_TotalCycles => stChopperWIP_Valve_Int.iTotalCycles,
    q_MaintCycles => stChopperWIP_Valve_Int.iMaintCycles,
    q_MaintenanceCall => stChopperWIP_Valve_Int.bMaintCall,
    q_State => stChopperWIP_Valve_Int.iState); // FB_ValveCtrl32
stChopperWIP_Valve_Int.bCmdOutWP := fbChopperWIP_Valve.q_Cmd;
OUT.bChopper_WIP_V807_5 := fbChopperWIP_Valve.q_Cmd;

// NETWORK 2
stChopperWIP_Valve_Int.bServiceMode := GV.stControl.bServiceMode;

// NETWORK 3
stChopperWIP_Valve_Int.arrInterlocks := F_ToArrInterlocks(In1 := NOT OUT.bChopper_Air_V807_6, In2 := TRUE, In3 := TRUE, In4 := TRUE, In5 := TRUE, In6 := TRUE, In7 := TRUE, In8 := TRUE);

// NETWORK 4
stChopperWIP_Valve_Int.arrAlarms := F_ToArrAlarms(In1 := fbChopperWIP_Valve.q_TimeoutHP, In2 := fbChopperWIP_Valve.q_TimeoutWP, In3 := fbChopperWIP_Valve.q_SensorsFlt, In4 := FALSE, In5 := FALSE, In6 := FALSE, In7 := FALSE, In8 := FALSE, AlarmsNOK => stChopperWIP_Valve_Int.bFault);

// NETWORK 5
stChopperWIP_Valve_Int.bCmdWP R= NOT stChopperWIP_Valve_Int.bServiceMode;

// NETWORK 6
END_ACTION

ACTION WIP_CleaningAir:
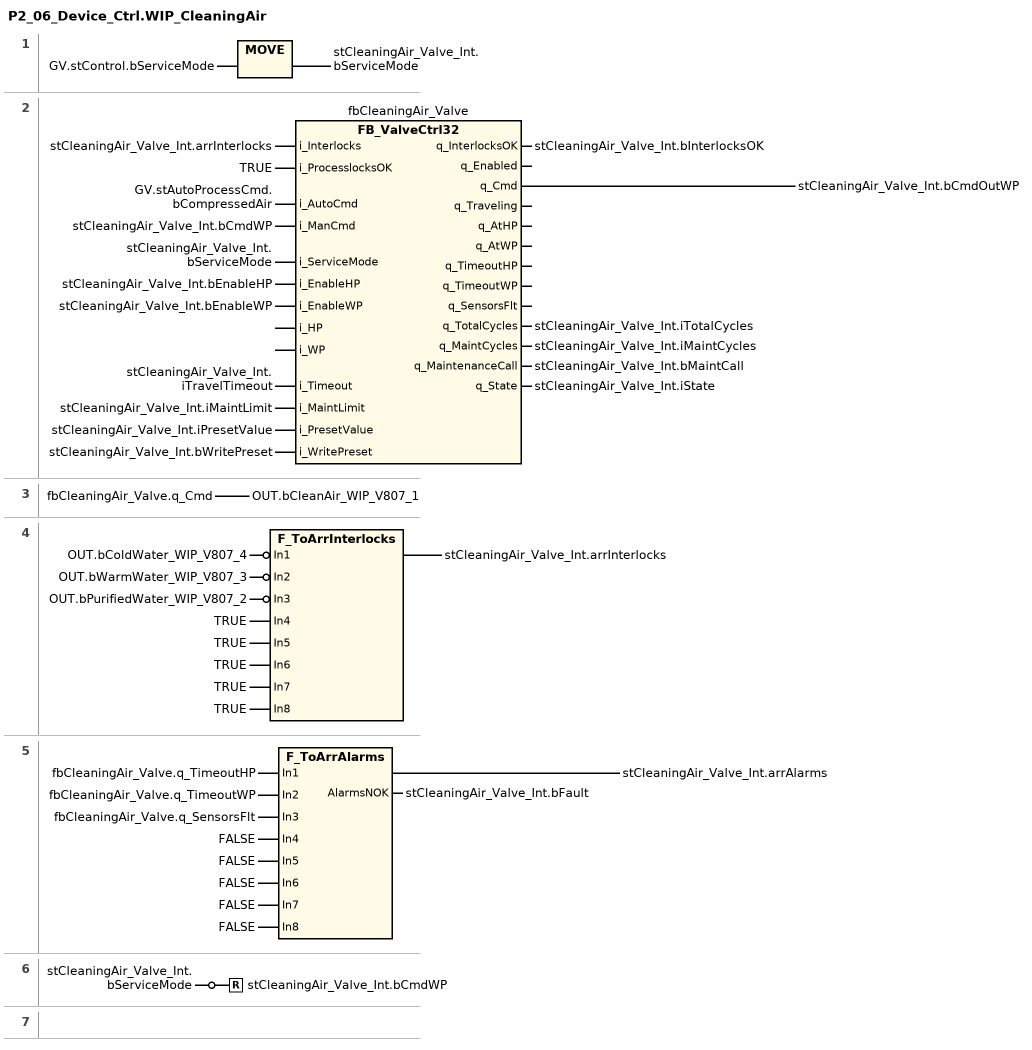
// NETWORK 1
stCleaningAir_Valve_Int.bServiceMode := GV.stControl.bServiceMode;

// NETWORK 2
fbCleaningAir_Valve(
    i_Interlocks := stCleaningAir_Valve_Int.arrInterlocks,
    i_ProcesslocksOK := TRUE,
    i_AutoCmd := GV.stAutoProcessCmd.bCompressedAir,
    i_ManCmd := stCleaningAir_Valve_Int.bCmdWP,
    i_ServiceMode := stCleaningAir_Valve_Int.bServiceMode,
    i_EnableHP := stCleaningAir_Valve_Int.bEnableHP,
    i_EnableWP := stCleaningAir_Valve_Int.bEnableWP,
    i_Timeout := stCleaningAir_Valve_Int.iTravelTimeout,
    i_MaintLimit := stCleaningAir_Valve_Int.iMaintLimit,
    i_PresetValue := stCleaningAir_Valve_Int.iPresetValue,
    i_WritePreset := stCleaningAir_Valve_Int.bWritePreset,
    q_InterlocksOK => stCleaningAir_Valve_Int.bInterlocksOK,
    q_TotalCycles => stCleaningAir_Valve_Int.iTotalCycles,
    q_MaintCycles => stCleaningAir_Valve_Int.iMaintCycles,
    q_MaintenanceCall => stCleaningAir_Valve_Int.bMaintCall,
    q_State => stCleaningAir_Valve_Int.iState); // FB_ValveCtrl32
stCleaningAir_Valve_Int.bCmdOutWP := fbCleaningAir_Valve.q_Cmd;

// NETWORK 3
OUT.bCleanAir_WIP_V807_1 := fbCleaningAir_Valve.q_Cmd;

// NETWORK 4
stCleaningAir_Valve_Int.arrInterlocks := F_ToArrInterlocks(In1 := NOT OUT.bColdWater_WIP_V807_4, In2 := NOT OUT.bWarmWater_WIP_V807_3, In3 := NOT OUT.bPurifiedWater_WIP_V807_2, In4 := TRUE, In5 := TRUE, In6 := TRUE, In7 := TRUE, In8 := TRUE);

// NETWORK 5
stCleaningAir_Valve_Int.arrAlarms := F_ToArrAlarms(In1 := fbCleaningAir_Valve.q_TimeoutHP, In2 := fbCleaningAir_Valve.q_TimeoutWP, In3 := fbCleaningAir_Valve.q_SensorsFlt, In4 := FALSE, In5 := FALSE, In6 := FALSE, In7 := FALSE, In8 := FALSE, AlarmsNOK => stCleaningAir_Valve_Int.bFault);

// NETWORK 6
stCleaningAir_Valve_Int.bCmdWP R= NOT stCleaningAir_Valve_Int.bServiceMode;

// NETWORK 7
END_ACTION

ACTION WIP_ColdWater:
